LIN {X -0.173,Y -453.003,Z 1528.498,A 0.000,B 0.000,C 90.000,E1 89.714} C_DIS
LIN {X -0.072,Y -440.256,Z 1528.488,A 0.000,B 0.000,C 90.000,E1 87.879} C_DIS
LIN {X 0.196,Y -427.118,Z 1528.478,A 0.000,B 0.000,C 90.000,E1 85.988} C_DIS
LIN {X -0.048,Y -412.183,Z 1528.466,A 0.000,B 0.000,C 90.000,E1 83.856} C_DIS
LIN {X -0.163,Y -397.400,Z 1528.453,A 0.000,B 0.000,C 90.000,E1 81.659} C_DIS
LIN {X -0.079,Y -377.981,Z 1528.436,A 0.000,B 0.000,C 90.000,E1 78.522} C_DIS
LIN {X 0.029,Y -364.705,Z 1528.423,A 0.000,B 0.000,C 90.000,E1 76.172} C_DIS
LIN {X -0.004,Y -351.765,Z 1528.410,A 0.000,B 0.000,C 90.000,E1 73.795} C_DIS
LIN {X 0.181,Y -340.593,Z 1528.398,A 0.000,B 0.000,C 90.000,E1 71.638} C_DIS
LIN {X 0.080,Y -323.637,Z 1528.379,A 0.000,B 0.000,C 90.000,E1 68.230} C_DIS
LIN {X 0.151,Y -311.879,Z 1528.365,A 0.000,B 0.000,C 90.000,E1 65.665} C_DIS
LIN {X 0.063,Y -300.644,Z 1528.350,A 0.000,B 0.000,C 90.000,E1 63.076} C_DIS
LIN {X -0.152,Y -289.519,Z 1528.336,A 0.000,B 0.000,C 90.000,E1 60.461} C_DIS
LIN {X -0.057,Y -280.084,Z 1528.323,A 0.000,B 0.000,C 90.000,E1 58.074} C_DIS
LIN {X -0.116,Y -270.752,Z 1528.309,A 0.000,B 0.000,C 90.000,E1 55.674} C_DIS
LIN {X 0.046,Y -259.191,Z 1528.292,A 0.000,B 0.000,C 90.000,E1 52.477} C_DIS
LIN {X -0.016,Y -248.168,Z 1528.274,A 0.000,B 0.000,C 90.000,E1 49.256} C_DIS
LIN {X -0.099,Y -237.990,Z 1528.255,A 0.000,B 0.000,C 90.000,E1 45.972} C_DIS
LIN {X 0.109,Y -229.786,Z 1528.239,A 0.000,B 0.000,C 90.000,E1 42.933} C_DIS
LIN {X -0.028,Y -222.332,Z 1528.222,A 0.000,B 0.000,C 90.000,E1 39.930} C_DIS
LIN {X -0.117,Y -215.621,Z 1528.205,A 0.000,B 0.000,C 90.000,E1 36.870} C_DIS
LIN {X 0.019,Y -209.646,Z 1528.187,A 0.000,B 0.000,C 90.000,E1 33.706} C_DIS
LIN {X 0.009,Y -204.410,Z 1528.170,A 0.000,B 0.000,C 90.000,E1 30.541} C_DIS
LIN {X -0.017,Y -198.622,Z 1528.147,A 0.000,B 0.000,C 90.000,E1 26.539} C_DIS
LIN {X 0.049,Y -193.675,Z 1528.125,A 0.000,B 0.000,C 90.000,E1 22.461} C_DIS
LIN {X 0.035,Y -189.499,Z 1528.102,A 0.000,B 0.000,C 90.000,E1 18.362} C_DIS
LIN {X -0.030,Y -185.543,Z 1528.074,A 0.000,B 0.000,C 90.000,E1 13.411} C_DIS
LIN {X -0.030,Y -182.509,Z 1528.047,A 0.000,B 0.000,C 90.000,E1 8.398} C_DIS
LIN {X 0.030,Y -180.027,Z 1528.005,A 0.000,B 0.000,C 90.000,E1 0.802} C_DIS
LIN {X -0.035,Y -180.270,Z 1527.965,A 0.000,B 0.000,C 90.000,E1 353.628} C_DIS
LIN {X -0.026,Y -182.584,Z 1527.927,A 0.000,B 0.000,C 90.000,E1 346.881} C_DIS
LIN {X 0.077,Y -185.773,Z 1527.899,A 0.000,B 0.000,C 90.000,E1 341.819} C_DIS
LIN {X 0.047,Y -189.339,Z 1527.876,A 0.000,B 0.000,C 90.000,E1 337.667} C_DIS
LIN {X -0.030,Y -193.881,Z 1527.853,A 0.000,B 0.000,C 90.000,E1 333.563} C_DIS
LIN {X 0.100,Y -198.154,Z 1527.835,A 0.000,B 0.000,C 90.000,E1 330.255} C_DIS
LIN {X 0.094,Y -204.384,Z 1527.813,A 0.000,B 0.000,C 90.000,E1 326.215} C_DIS
LIN {X -0.012,Y -210.151,Z 1527.795,A 0.000,B 0.000,C 90.000,E1 323.050} C_DIS
LIN {X -0.059,Y -216.737,Z 1527.777,A 0.000,B 0.000,C 90.000,E1 319.908} C_DIS
LIN {X 0.005,Y -224.124,Z 1527.760,A 0.000,B 0.000,C 90.000,E1 316.782} C_DIS
LIN {X 0.043,Y -233.399,Z 1527.741,A 0.000,B 0.000,C 90.000,E1 313.338} C_DIS
LIN {X 0.126,Y -240.429,Z 1527.728,A 0.000,B 0.000,C 90.000,E1 311.067} C_DIS
LIN {X -0.137,Y -248.431,Z 1527.716,A 0.000,B 0.000,C 90.000,E1 308.910} C_DIS
LIN {X -0.087,Y -255.980,Z 1527.706,A 0.000,B 0.000,C 90.000,E1 307.076} C_DIS
LIN {X 0.099,Y -262.847,Z 1527.698,A 0.000,B 0.000,C 90.000,E1 305.598} C_DIS
LIN {X 0.009,Y -270.418,Z 1527.690,A 0.000,B 0.000,C 90.000,E1 304.199} C_DIS
LIN {X -0.047,Y -280.857,Z 1527.680,A 0.000,B 0.000,C 90.000,E1 302.467} C_DIS
LIN {X -0.034,Y -297.223,Z 1527.667,A 0.000,B 0.000,C 90.000,E1 300.079} C_DIS
LIN {X 0.000,Y -317.615,Z 1527.652,A 0.000,B 0.000,C 90.000,E1 297.436} C_DIS
LIN {X 0.091,Y -333.573,Z 1527.642,A 0.000,B 0.000,C 90.000,E1 295.540} C_DIS
LIN {X -0.050,Y -349.616,Z 1527.632,A 0.000,B 0.000,C 90.000,E1 293.770} C_DIS
LIN {X 0.136,Y -365.761,Z 1527.622,A 0.000,B 0.000,C 90.000,E1 292.025} C_DIS
LIN {X -0.085,Y -378.909,Z 1527.615,A 0.000,B 0.000,C 90.000,E1 290.663} C_DIS
LIN {X -0.010,Y -386.648,Z 1527.610,A 0.000,B 0.000,C 90.000,E1 289.812} C_DIS
LIN {X 0.039,Y -396.456,Z 1527.604,A 0.000,B 0.000,C 90.000,E1 288.671} C_DIS
LIN {X 0.076,Y -403.212,Z 1527.599,A 0.000,B 0.000,C 90.000,E1 287.819} C_DIS
LIN {X 0.046,Y -409.350,Z 1527.594,A 0.000,B 0.000,C 90.000,E1 286.985} C_DIS
LIN {X 0.081,Y -414.751,Z 1527.590,A 0.000,B 0.000,C 90.000,E1 286.150} C_DIS
LIN {X -0.242,Y -419.471,Z 1527.585,A 0.000,B 0.000,C 90.000,E1 285.371} C_DIS
LIN {X -0.119,Y -423.315,Z 1527.581,A 0.000,B 0.000,C 90.000,E1 284.537} C_DIS
LIN {X 0.035,Y -426.460,Z 1527.576,A 0.000,B 0.000,C 90.000,E1 283.703} C_DIS
LIN {X -0.057,Y -428.128,Z 1527.573,A 0.000,B 0.000,C 90.000,E1 283.175} C_DIS
LIN {X -0.138,Y -429.417,Z 1527.570,A 0.000,B 0.000,C 90.000,E1 282.647} C_DIS
LIN {X 0.213,Y -430.220,Z 1527.567,A 0.000,B 0.000,C 90.000,E1 282.063} C_DIS
LIN {X 0.150,Y -430.594,Z 1527.564,A 0.000,B 0.000,C 90.000,E1 281.535} C_DIS
LIN {X 0.091,Y -430.469,Z 1527.561,A 0.000,B 0.000,C 90.000,E1 281.007} C_DIS
LIN {X -0.045,Y -429.811,Z 1527.558,A 0.000,B 0.000,C 90.000,E1 280.489} C_DIS
LIN {X -0.103,Y -428.580,Z 1527.555,A 0.000,B 0.000,C 90.000,E1 279.962} C_DIS
LIN {X -0.167,Y -426.752,Z 1527.552,A 0.000,B 0.000,C 90.000,E1 279.434} C_DIS
LIN {X 0.112,Y -424.208,Z 1527.549,A 0.000,B 0.000,C 90.000,E1 278.859} C_DIS
LIN {X -0.042,Y -420.783,Z 1527.546,A 0.000,B 0.000,C 90.000,E1 278.341} C_DIS
LIN {X 0.111,Y -418.773,Z 1527.545,A 0.000,B 0.000,C 90.000,E1 278.049} C_DIS
LIN {X -0.068,Y -413.948,Z 1527.542,A 0.000,B 0.000,C 90.000,E1 277.530} C_DIS
LIN {X 0.070,Y -411.225,Z 1527.540,A 0.000,B 0.000,C 90.000,E1 277.239} C_DIS
LIN {X 0.063,Y -405.102,Z 1527.537,A 0.000,B 0.000,C 90.000,E1 276.720} C_DIS
LIN {X 0.110,Y -399.086,Z 1527.535,A 0.000,B 0.000,C 90.000,E1 276.258} C_DIS
LIN {X 0.027,Y -392.632,Z 1527.533,A 0.000,B 0.000,C 90.000,E1 275.853} C_DIS
LIN {X -0.142,Y -386.213,Z 1527.531,A 0.000,B 0.000,C 90.000,E1 275.511} C_DIS
LIN {X 0.106,Y -376.409,Z 1527.528,A 0.000,B 0.000,C 90.000,E1 274.992} C_DIS
LIN {X -0.035,Y -366.667,Z 1527.526,A 0.000,B 0.000,C 90.000,E1 274.588} C_DIS
LIN {X -0.112,Y -351.054,Z 1527.522,A 0.000,B 0.000,C 90.000,E1 273.955} C_DIS
LIN {X 0.037,Y -341.268,Z 1527.520,A 0.000,B 0.000,C 90.000,E1 273.555} C_DIS
LIN {X 0.087,Y -331.254,Z 1527.518,A 0.000,B 0.000,C 90.000,E1 273.212} C_DIS
LIN {X 0.142,Y -317.896,Z 1527.516,A 0.000,B 0.000,C 90.000,E1 272.808} C_DIS
LIN {X -0.021,Y -306.821,Z 1527.514,A 0.000,B 0.000,C 90.000,E1 272.579} C_DIS
LIN {X 0.106,Y -295.216,Z 1527.513,A 0.000,B 0.000,C 90.000,E1 272.350} C_DIS
LIN {X 0.098,Y -281.912,Z 1527.512,A 0.000,B 0.000,C 90.000,E1 272.178} C_DIS
LIN {X 0.024,Y -268.089,Z 1527.512,A 0.000,B 0.000,C 90.000,E1 272.121} C_DIS
LIN {X -0.008,Y -265.982,Z 1527.512,A 0.000,B 0.000,C 90.000,E1 272.121} C_DIS
LIN {X -0.027,Y -181.243,Z 1527.512,A 0.000,B 0.000,C 90.000,E1 272.121} C_DIS
LIN {X 0.068,Y -181.571,Z 1527.500,A 0.000,B 0.000,C 90.000,E1 270.057} C_DIS
LIN {X 0.056,Y -180.867,Z 1527.472,A 0.000,B 0.000,C 90.000,E1 265.008} C_DIS
LIN {X -0.067,Y -178.983,Z 1527.444,A 0.000,B 0.000,C 90.000,E1 259.982} C_DIS
LIN {X -0.056,Y -177.955,Z 1527.435,A 0.000,B 0.000,C 90.000,E1 258.285} C_DIS
LIN {X -0.037,Y -175.597,Z 1527.411,A 0.000,B 0.000,C 90.000,E1 254.031} C_DIS
LIN {X -0.023,Y -172.320,Z 1527.387,A 0.000,B 0.000,C 90.000,E1 249.752} C_DIS
LIN {X -0.045,Y -171.799,Z 1527.383,A 0.000,B 0.000,C 90.000,E1 248.901} C_DIS
LIN {X -0.007,Y -169.472,Z 1527.368,A 0.000,B 0.000,C 90.000,E1 246.305} C_DIS
LIN {X 0.048,Y -166.799,Z 1527.349,A 0.000,B 0.000,C 90.000,E1 242.820} C_DIS
LIN {X 0.043,Y -162.779,Z 1527.325,A 0.000,B 0.000,C 90.000,E1 238.456} C_DIS
LIN {X 0.019,Y -161.468,Z 1527.315,A 0.000,B 0.000,C 90.000,E1 236.707} C_DIS
LIN {X 0.059,Y -157.464,Z 1527.291,A 0.000,B 0.000,C 90.000,E1 232.271} C_DIS
LIN {X -0.008,Y -155.476,Z 1527.276,A 0.000,B 0.000,C 90.000,E1 229.622} C_DIS
LIN {X -0.074,Y -151.787,Z 1527.251,A 0.000,B 0.000,C 90.000,E1 225.162} C_DIS
LIN {X -0.061,Y -149.994,Z 1527.236,A 0.000,B 0.000,C 90.000,E1 222.447} C_DIS
LIN {X -0.030,Y -146.824,Z 1527.210,A 0.000,B 0.000,C 90.000,E1 217.890} C_DIS
LIN {X 0.076,Y -145.404,Z 1527.195,A 0.000,B 0.000,C 90.000,E1 215.105} C_DIS
LIN {X -0.007,Y -142.836,Z 1527.170,A 0.000,B 0.000,C 90.000,E1 210.541} C_DIS
LIN {X -0.077,Y -141.450,Z 1527.149,A 0.000,B 0.000,C 90.000,E1 206.873} C_DIS
LIN {X -0.036,Y -139.371,Z 1527.113,A 0.000,B 0.000,C 90.000,E1 200.355} C_DIS
LIN {X 0.038,Y -138.820,Z 1527.097,A 0.000,B 0.000,C 90.000,E1 197.528} C_DIS
LIN {X -0.005,Y -138.352,Z 1527.056,A 0.000,B 0.000,C 90.000,E1 190.074} C_DIS
LIN {X -0.033,Y -139.534,Z 1527.004,A 0.000,B 0.000,C 90.000,E1 180.745} C_DIS
LIN {X 0.060,Y -141.219,Z 1526.973,A 0.000,B 0.000,C 90.000,E1 175.122} C_DIS
LIN {X 0.019,Y -142.593,Z 1526.958,A 0.000,B 0.000,C 90.000,E1 172.356} C_DIS
LIN {X -0.027,Y -144.894,Z 1526.932,A 0.000,B 0.000,C 90.000,E1 167.757} C_DIS
LIN {X -0.074,Y -147.522,Z 1526.911,A 0.000,B 0.000,C 90.000,E1 164.102} C_DIS
LIN {X 0.000,Y -150.118,Z 1526.891,A 0.000,B 0.000,C 90.000,E1 160.423} C_DIS
LIN {X 0.012,Y -153.479,Z 1526.871,A 0.000,B 0.000,C 90.000,E1 156.794} C_DIS
LIN {X 0.076,Y -157.842,Z 1526.846,A 0.000,B 0.000,C 90.000,E1 152.281} C_DIS
LIN {X 0.032,Y -162.128,Z 1526.826,A 0.000,B 0.000,C 90.000,E1 148.742} C_DIS
LIN {X 0.011,Y -166.330,Z 1526.807,A 0.000,B 0.000,C 90.000,E1 145.229} C_DIS
LIN {X 0.018,Y -171.347,Z 1526.787,A 0.000,B 0.000,C 90.000,E1 141.743} C_DIS
LIN {X -0.054,Y -176.251,Z 1526.768,A 0.000,B 0.000,C 90.000,E1 138.324} C_DIS
LIN {X 0.064,Y -180.533,Z 1526.754,A 0.000,B 0.000,C 90.000,E1 135.729} C_DIS
LIN {X 0.043,Y -185.936,Z 1526.735,A 0.000,B 0.000,C 90.000,E1 132.366} C_DIS
LIN {X -0.021,Y -190.566,Z 1526.722,A 0.000,B 0.000,C 90.000,E1 129.886} C_DIS
LIN {X 0.009,Y -196.316,Z 1526.703,A 0.000,B 0.000,C 90.000,E1 126.583} C_DIS
LIN {X 0.087,Y -201.115,Z 1526.690,A 0.000,B 0.000,C 90.000,E1 124.119} C_DIS
LIN {X 0.060,Y -202.556,Z 1526.685,A 0.000,B 0.000,C 90.000,E1 123.293} C_DIS
LIN {X 0.042,Y -317.227,Z 1526.685,A 0.000,B 0.000,C 90.000,E1 123.293} C_DIS
LIN {X -0.114,Y -318.999,Z 1526.685,A 0.000,B 0.000,C 90.000,E1 123.293} C_DIS
LIN {X 0.003,Y -323.259,Z 1526.684,A 0.000,B 0.000,C 90.000,E1 123.086} C_DIS
LIN {X 0.122,Y -325.660,Z 1526.683,A 0.000,B 0.000,C 90.000,E1 122.880} C_DIS
LIN {X -0.092,Y -328.932,Z 1526.681,A 0.000,B 0.000,C 90.000,E1 122.546} C_DIS
LIN {X 0.077,Y -330.854,Z 1526.679,A 0.000,B 0.000,C 90.000,E1 122.212} C_DIS
LIN {X -0.033,Y -332.352,Z 1526.677,A 0.000,B 0.000,C 90.000,E1 121.926} C_DIS
LIN {X 0.120,Y -346.150,Z 1526.658,A 0.000,B 0.000,C 90.000,E1 118.487} C_DIS
LIN {X 0.015,Y -358.945,Z 1526.643,A 0.000,B 0.000,C 90.000,E1 115.771} C_DIS
LIN {X 0.137,Y -373.256,Z 1526.628,A 0.000,B 0.000,C 90.000,E1 113.078} C_DIS
LIN {X -0.112,Y -387.354,Z 1526.615,A 0.000,B 0.000,C 90.000,E1 110.791} C_DIS
LIN {X 0.084,Y -402.848,Z 1526.603,A 0.000,B 0.000,C 90.000,E1 108.489} C_DIS
LIN {X 0.165,Y -419.844,Z 1526.590,A 0.000,B 0.000,C 90.000,E1 106.260} C_DIS
LIN {X 0.012,Y -438.465,Z 1526.578,A 0.000,B 0.000,C 90.000,E1 104.120} C_DIS
LIN {X 0.039,Y -458.333,Z 1526.567,A 0.000,B 0.000,C 90.000,E1 102.063} C_DIS
LIN {X -0.147,Y -478.777,Z 1526.557,A 0.000,B 0.000,C 90.000,E1 100.197} C_DIS
LIN {X -0.161,Y -491.735,Z 1526.550,A 0.000,B 0.000,C 90.000,E1 99.095} C_DIS
LIN {X -0.031,Y -493.741,Z 1526.549,A 0.000,B 0.000,C 90.000,E1 98.859} C_DIS
LIN {X 0.099,Y -495.273,Z 1526.548,A 0.000,B 0.000,C 90.000,E1 98.624} C_DIS
LIN {X -0.061,Y -496.569,Z 1526.547,A 0.000,B 0.000,C 90.000,E1 98.398} C_DIS
LIN {X -0.149,Y -497.517,Z 1526.545,A 0.000,B 0.000,C 90.000,E1 98.163} C_DIS
LIN {X 0.114,Y -498.549,Z 1526.542,A 0.000,B 0.000,C 90.000,E1 97.644} C_DIS
LIN {X -0.110,Y -498.564,Z 1526.540,A 0.000,B 0.000,C 90.000,E1 97.182} C_DIS
LIN {X 0.166,Y -497.568,Z 1526.537,A 0.000,B 0.000,C 90.000,E1 96.663} C_DIS
LIN {X 0.084,Y -496.645,Z 1526.536,A 0.000,B 0.000,C 90.000,E1 96.429} C_DIS
LIN {X -0.052,Y -495.385,Z 1526.534,A 0.000,B 0.000,C 90.000,E1 96.201} C_DIS
LIN {X -0.132,Y -482.564,Z 1526.523,A 0.000,B 0.000,C 90.000,E1 94.245} C_DIS
LIN {X 0.031,Y -474.878,Z 1526.517,A 0.000,B 0.000,C 90.000,E1 92.980} C_DIS
LIN {X -0.148,Y -465.003,Z 1526.508,A 0.000,B 0.000,C 90.000,E1 91.489} C_DIS
LIN {X 0.185,Y -456.365,Z 1526.501,A 0.000,B 0.000,C 90.000,E1 90.172} C_DIS
LIN {X -0.066,Y -447.398,Z 1526.494,A 0.000,B 0.000,C 90.000,E1 88.912} C_DIS
LIN {X 0.019,Y -438.249,Z 1526.487,A 0.000,B 0.000,C 90.000,E1 87.593} C_DIS
LIN {X -0.160,Y -425.115,Z 1526.476,A 0.000,B 0.000,C 90.000,E1 85.755} C_DIS
LIN {X -0.064,Y -410.273,Z 1526.464,A 0.000,B 0.000,C 90.000,E1 83.571} C_DIS
LIN {X -0.154,Y -393.712,Z 1526.450,A 0.000,B 0.000,C 90.000,E1 81.084} C_DIS
LIN {X -0.141,Y -376.233,Z 1526.434,A 0.000,B 0.000,C 90.000,E1 78.229} C_DIS
LIN {X -0.074,Y -363.041,Z 1526.422,A 0.000,B 0.000,C 90.000,E1 75.880} C_DIS
LIN {X -0.086,Y -351.730,Z 1526.410,A 0.000,B 0.000,C 90.000,E1 73.795} C_DIS
LIN {X 0.101,Y -340.554,Z 1526.398,A 0.000,B 0.000,C 90.000,E1 71.638} C_DIS
LIN {X 0.002,Y -323.597,Z 1526.379,A 0.000,B 0.000,C 90.000,E1 68.230} C_DIS
LIN {X -0.002,Y -310.395,Z 1526.363,A 0.000,B 0.000,C 90.000,E1 65.357} C_DIS
LIN {X 0.011,Y -299.185,Z 1526.349,A 0.000,B 0.000,C 90.000,E1 62.743} C_DIS
LIN {X 0.018,Y -288.141,Z 1526.334,A 0.000,B 0.000,C 90.000,E1 60.078} C_DIS
LIN {X -0.019,Y -278.750,Z 1526.321,A 0.000,B 0.000,C 90.000,E1 57.709} C_DIS
LIN {X -0.170,Y -268.179,Z 1526.305,A 0.000,B 0.000,C 90.000,E1 54.975} C_DIS
LIN {X 0.030,Y -258.026,Z 1526.290,A 0.000,B 0.000,C 90.000,E1 52.110} C_DIS
LIN {X 0.102,Y -247.111,Z 1526.271,A 0.000,B 0.000,C 90.000,E1 48.852} C_DIS
LIN {X -0.152,Y -238.144,Z 1526.255,A 0.000,B 0.000,C 90.000,E1 45.972} C_DIS
LIN {X 0.068,Y -229.958,Z 1526.239,A 0.000,B 0.000,C 90.000,E1 42.933} C_DIS
LIN {X -0.064,Y -222.521,Z 1526.222,A 0.000,B 0.000,C 90.000,E1 39.930} C_DIS
LIN {X 0.026,Y -215.851,Z 1526.205,A 0.000,B 0.000,C 90.000,E1 36.824} C_DIS
LIN {X -0.004,Y -209.917,Z 1526.187,A 0.000,B 0.000,C 90.000,E1 33.706} C_DIS
LIN {X -0.006,Y -204.679,Z 1526.170,A 0.000,B 0.000,C 90.000,E1 30.541} C_DIS
LIN {X -0.024,Y -198.893,Z 1526.147,A 0.000,B 0.000,C 90.000,E1 26.539} C_DIS
LIN {X 0.051,Y -193.952,Z 1526.125,A 0.000,B 0.000,C 90.000,E1 22.461} C_DIS
LIN {X 0.045,Y -189.771,Z 1526.102,A 0.000,B 0.000,C 90.000,E1 18.362} C_DIS
LIN {X -0.010,Y -185.781,Z 1526.074,A 0.000,B 0.000,C 90.000,E1 13.411} C_DIS
LIN {X -0.092,Y -182.340,Z 1526.042,A 0.000,B 0.000,C 90.000,E1 7.587} C_DIS
LIN {X -0.032,Y -180.199,Z 1525.997,A 0.000,B 0.000,C 90.000,E1 359.542} C_DIS
LIN {X 0.050,Y -180.694,Z 1525.960,A 0.000,B 0.000,C 90.000,E1 352.761} C_DIS
LIN {X -0.023,Y -183.276,Z 1525.922,A 0.000,B 0.000,C 90.000,E1 346.047} C_DIS
LIN {X -0.068,Y -186.654,Z 1525.895,A 0.000,B 0.000,C 90.000,E1 341.040} C_DIS
LIN {X -0.012,Y -190.368,Z 1525.871,A 0.000,B 0.000,C 90.000,E1 336.869} C_DIS
LIN {X 0.020,Y -195.079,Z 1525.849,A 0.000,B 0.000,C 90.000,E1 332.743} C_DIS
LIN {X 0.050,Y -200.690,Z 1525.826,A 0.000,B 0.000,C 90.000,E1 328.663} C_DIS
LIN {X -0.041,Y -205.912,Z 1525.808,A 0.000,B 0.000,C 90.000,E1 325.468} C_DIS
LIN {X 0.008,Y -211.870,Z 1525.790,A 0.000,B 0.000,C 90.000,E1 322.271} C_DIS
LIN {X -0.026,Y -218.636,Z 1525.773,A 0.000,B 0.000,C 90.000,E1 319.138} C_DIS
LIN {X 0.011,Y -227.200,Z 1525.754,A 0.000,B 0.000,C 90.000,E1 315.648} C_DIS
LIN {X 0.029,Y -235.753,Z 1525.737,A 0.000,B 0.000,C 90.000,E1 312.609} C_DIS
LIN {X -0.008,Y -243.086,Z 1525.724,A 0.000,B 0.000,C 90.000,E1 310.378} C_DIS
LIN {X -0.032,Y -251.392,Z 1525.712,A 0.000,B 0.000,C 90.000,E1 308.177} C_DIS
LIN {X 0.041,Y -257.616,Z 1525.704,A 0.000,B 0.000,C 90.000,E1 306.710} C_DIS
LIN {X -0.070,Y -266.486,Z 1525.694,A 0.000,B 0.000,C 90.000,E1 304.945} C_DIS
LIN {X 0.035,Y -276.442,Z 1525.684,A 0.000,B 0.000,C 90.000,E1 303.166} C_DIS
LIN {X -0.085,Y -287.502,Z 1525.675,A 0.000,B 0.000,C 90.000,E1 301.465} C_DIS
LIN {X -0.008,Y -309.538,Z 1525.658,A 0.000,B 0.000,C 90.000,E1 298.437} C_DIS
LIN {X -0.082,Y -330.555,Z 1525.644,A 0.000,B 0.000,C 90.000,E1 295.924} C_DIS
LIN {X 0.157,Y -349.448,Z 1525.632,A 0.000,B 0.000,C 90.000,E1 293.770} C_DIS
LIN {X 0.030,Y -365.620,Z 1525.623,A 0.000,B 0.000,C 90.000,E1 292.078} C_DIS
LIN {X 0.051,Y -378.769,Z 1525.615,A 0.000,B 0.000,C 90.000,E1 290.684} C_DIS
LIN {X -0.088,Y -386.496,Z 1525.610,A 0.000,B 0.000,C 90.000,E1 289.866} C_DIS
LIN {X -0.088,Y -393.952,Z 1525.606,A 0.000,B 0.000,C 90.000,E1 289.014} C_DIS
LIN {X -0.212,Y -401.000,Z 1525.601,A 0.000,B 0.000,C 90.000,E1 288.181} C_DIS
LIN {X -0.141,Y -407.348,Z 1525.596,A 0.000,B 0.000,C 90.000,E1 287.330} C_DIS
LIN {X -0.138,Y -413.082,Z 1525.592,A 0.000,B 0.000,C 90.000,E1 286.496} C_DIS
LIN {X 0.203,Y -416.536,Z 1525.589,A 0.000,B 0.000,C 90.000,E1 285.898} C_DIS
LIN {X 0.053,Y -419.609,Z 1525.585,A 0.000,B 0.000,C 90.000,E1 285.371} C_DIS
LIN {X 0.180,Y -423.507,Z 1525.581,A 0.000,B 0.000,C 90.000,E1 284.537} C_DIS
LIN {X 0.077,Y -425.750,Z 1525.578,A 0.000,B 0.000,C 90.000,E1 284.008} C_DIS
LIN {X -0.163,Y -428.421,Z 1525.573,A 0.000,B 0.000,C 90.000,E1 283.231} C_DIS
LIN {X 0.176,Y -429.747,Z 1525.570,A 0.000,B 0.000,C 90.000,E1 282.647} C_DIS
LIN {X 0.108,Y -430.664,Z 1525.567,A 0.000,B 0.000,C 90.000,E1 282.119} C_DIS
LIN {X 0.047,Y -431.055,Z 1525.564,A 0.000,B 0.000,C 90.000,E1 281.591} C_DIS
LIN {X -0.093,Y -431.020,Z 1525.561,A 0.000,B 0.000,C 90.000,E1 281.074} C_DIS
LIN {X -0.146,Y -430.406,Z 1525.558,A 0.000,B 0.000,C 90.000,E1 280.546} C_DIS
LIN {X 0.222,Y -429.247,Z 1525.556,A 0.000,B 0.000,C 90.000,E1 279.962} C_DIS
LIN {X 0.091,Y -427.504,Z 1525.552,A 0.000,B 0.000,C 90.000,E1 279.443} C_DIS
LIN {X 0.022,Y -425.035,Z 1525.550,A 0.000,B 0.000,C 90.000,E1 278.916} C_DIS
LIN {X -0.127,Y -421.724,Z 1525.547,A 0.000,B 0.000,C 90.000,E1 278.398} C_DIS
LIN {X 0.028,Y -419.779,Z 1525.545,A 0.000,B 0.000,C 90.000,E1 278.106} C_DIS
LIN {X -0.144,Y -415.081,Z 1525.542,A 0.000,B 0.000,C 90.000,E1 277.587} C_DIS
LIN {X -0.223,Y -409.526,Z 1525.539,A 0.000,B 0.000,C 90.000,E1 277.068} C_DIS
LIN {X 0.002,Y -403.518,Z 1525.536,A 0.000,B 0.000,C 90.000,E1 276.549} C_DIS
LIN {X 0.155,Y -397.292,Z 1525.534,A 0.000,B 0.000,C 90.000,E1 276.087} C_DIS
LIN {X -0.180,Y -390.890,Z 1525.532,A 0.000,B 0.000,C 90.000,E1 275.739} C_DIS
LIN {X 0.156,Y -384.382,Z 1525.530,A 0.000,B 0.000,C 90.000,E1 275.334} C_DIS
LIN {X 0.051,Y -374.399,Z 1525.527,A 0.000,B 0.000,C 90.000,E1 274.878} C_DIS
LIN {X -0.149,Y -358.593,Z 1525.523,A 0.000,B 0.000,C 90.000,E1 274.245} C_DIS
LIN {X -0.071,Y -345.966,Z 1525.521,A 0.000,B 0.000,C 90.000,E1 273.726} C_DIS
LIN {X -0.158,Y -335.860,Z 1525.519,A 0.000,B 0.000,C 90.000,E1 273.383} C_DIS
LIN {X 0.153,Y -322.648,Z 1525.516,A 0.000,B 0.000,C 90.000,E1 272.922} C_DIS
LIN {X -0.096,Y -311.980,Z 1525.515,A 0.000,B 0.000,C 90.000,E1 272.694} C_DIS
LIN {X -0.107,Y -300.382,Z 1525.514,A 0.000,B 0.000,C 90.000,E1 272.465} C_DIS
LIN {X 0.139,Y -287.899,Z 1525.513,A 0.000,B 0.000,C 90.000,E1 272.236} C_DIS
LIN {X -0.076,Y -276.839,Z 1525.512,A 0.000,B 0.000,C 90.000,E1 272.178} C_DIS
LIN {X 0.005,Y -265.525,Z 1525.512,A 0.000,B 0.000,C 90.000,E1 272.121} C_DIS
LIN {X -0.018,Y -181.244,Z 1525.512,A 0.000,B 0.000,C 90.000,E1 272.121} C_DIS
LIN {X -0.082,Y -181.572,Z 1525.500,A 0.000,B 0.000,C 90.000,E1 270.115} C_DIS
LIN {X 0.086,Y -180.870,Z 1525.472,A 0.000,B 0.000,C 90.000,E1 265.008} C_DIS
LIN {X -0.037,Y -178.985,Z 1525.444,A 0.000,B 0.000,C 90.000,E1 259.982} C_DIS
LIN {X -0.025,Y -177.962,Z 1525.435,A 0.000,B 0.000,C 90.000,E1 258.285} C_DIS
LIN {X -0.006,Y -175.604,Z 1525.411,A 0.000,B 0.000,C 90.000,E1 254.031} C_DIS
LIN {X 0.006,Y -172.328,Z 1525.388,A 0.000,B 0.000,C 90.000,E1 249.752} C_DIS
LIN {X -0.015,Y -171.804,Z 1525.383,A 0.000,B 0.000,C 90.000,E1 248.901} C_DIS
LIN {X -0.008,Y -170.264,Z 1525.373,A 0.000,B 0.000,C 90.000,E1 247.177} C_DIS
LIN {X -0.071,Y -166.807,Z 1525.349,A 0.000,B 0.000,C 90.000,E1 242.871} C_DIS
LIN {X 0.072,Y -162.788,Z 1525.325,A 0.000,B 0.000,C 90.000,E1 238.456} C_DIS
LIN {X 0.047,Y -161.476,Z 1525.315,A 0.000,B 0.000,C 90.000,E1 236.707} C_DIS
LIN {X -0.037,Y -157.471,Z 1525.291,A 0.000,B 0.000,C 90.000,E1 232.316} C_DIS
LIN {X 0.020,Y -155.486,Z 1525.276,A 0.000,B 0.000,C 90.000,E1 229.622} C_DIS
LIN {X -0.048,Y -151.794,Z 1525.251,A 0.000,B 0.000,C 90.000,E1 225.162} C_DIS
LIN {X -0.034,Y -150.003,Z 1525.236,A 0.000,B 0.000,C 90.000,E1 222.447} C_DIS
LIN {X -0.003,Y -146.830,Z 1525.210,A 0.000,B 0.000,C 90.000,E1 217.890} C_DIS
LIN {X -0.016,Y -145.411,Z 1525.195,A 0.000,B 0.000,C 90.000,E1 215.152} C_DIS
LIN {X 0.019,Y -142.841,Z 1525.170,A 0.000,B 0.000,C 90.000,E1 210.541} C_DIS
LIN {X -0.050,Y -141.455,Z 1525.149,A 0.000,B 0.000,C 90.000,E1 206.873} C_DIS
LIN {X -0.011,Y -139.373,Z 1525.113,A 0.000,B 0.000,C 90.000,E1 200.355} C_DIS
LIN {X -0.068,Y -138.822,Z 1525.098,A 0.000,B 0.000,C 90.000,E1 197.583} C_DIS
LIN {X 0.020,Y -138.353,Z 1525.056,A 0.000,B 0.000,C 90.000,E1 190.074} C_DIS
LIN {X -0.007,Y -139.533,Z 1525.004,A 0.000,B 0.000,C 90.000,E1 180.745} C_DIS
LIN {X -0.054,Y -141.214,Z 1524.973,A 0.000,B 0.000,C 90.000,E1 175.179} C_DIS
LIN {X 0.046,Y -142.588,Z 1524.958,A 0.000,B 0.000,C 90.000,E1 172.356} C_DIS
LIN {X 0.000,Y -144.887,Z 1524.932,A 0.000,B 0.000,C 90.000,E1 167.757} C_DIS
LIN {X -0.047,Y -147.515,Z 1524.912,A 0.000,B 0.000,C 90.000,E1 164.102} C_DIS
LIN {X 0.027,Y -150.109,Z 1524.891,A 0.000,B 0.000,C 90.000,E1 160.423} C_DIS
LIN {X 0.040,Y -153.468,Z 1524.871,A 0.000,B 0.000,C 90.000,E1 156.794} C_DIS
LIN {X 0.031,Y -157.832,Z 1524.846,A 0.000,B 0.000,C 90.000,E1 152.308} C_DIS
LIN {X 0.060,Y -162.115,Z 1524.826,A 0.000,B 0.000,C 90.000,E1 148.742} C_DIS
LIN {X -0.054,Y -166.317,Z 1524.807,A 0.000,B 0.000,C 90.000,E1 145.261} C_DIS
LIN {X 0.048,Y -171.335,Z 1524.788,A 0.000,B 0.000,C 90.000,E1 141.743} C_DIS
LIN {X -0.024,Y -176.236,Z 1524.768,A 0.000,B 0.000,C 90.000,E1 138.324} C_DIS
LIN {X 0.095,Y -180.516,Z 1524.754,A 0.000,B 0.000,C 90.000,E1 135.729} C_DIS
LIN {X 0.075,Y -185.919,Z 1524.735,A 0.000,B 0.000,C 90.000,E1 132.366} C_DIS
LIN {X 0.011,Y -190.548,Z 1524.722,A 0.000,B 0.000,C 90.000,E1 129.886} C_DIS
LIN {X 0.042,Y -196.299,Z 1524.703,A 0.000,B 0.000,C 90.000,E1 126.583} C_DIS
LIN {X 0.120,Y -201.098,Z 1524.690,A 0.000,B 0.000,C 90.000,E1 124.119} C_DIS
LIN {X -0.119,Y -202.506,Z 1524.685,A 0.000,B 0.000,C 90.000,E1 123.372} C_DIS
LIN {X 0.217,Y -317.322,Z 1524.685,A 0.000,B 0.000,C 90.000,E1 123.293} C_DIS
LIN {X -0.062,Y -319.730,Z 1524.685,A 0.000,B 0.000,C 90.000,E1 123.293} C_DIS
LIN {X 0.055,Y -323.481,Z 1524.684,A 0.000,B 0.000,C 90.000,E1 123.086} C_DIS
LIN {X 0.175,Y -325.777,Z 1524.683,A 0.000,B 0.000,C 90.000,E1 122.880} C_DIS
LIN {X -0.039,Y -328.959,Z 1524.681,A 0.000,B 0.000,C 90.000,E1 122.546} C_DIS
LIN {X 0.097,Y -330.873,Z 1524.679,A 0.000,B 0.000,C 90.000,E1 122.212} C_DIS
LIN {X -0.049,Y -332.363,Z 1524.677,A 0.000,B 0.000,C 90.000,E1 121.926} C_DIS
LIN {X -0.059,Y -344.809,Z 1524.660,A 0.000,B 0.000,C 90.000,E1 118.821} C_DIS
LIN {X 0.123,Y -357.440,Z 1524.645,A 0.000,B 0.000,C 90.000,E1 116.052} C_DIS
LIN {X 0.024,Y -371.581,Z 1524.630,A 0.000,B 0.000,C 90.000,E1 113.387} C_DIS
LIN {X 0.088,Y -385.514,Z 1524.617,A 0.000,B 0.000,C 90.000,E1 111.046} C_DIS
LIN {X 0.001,Y -400.829,Z 1524.604,A 0.000,B 0.000,C 90.000,E1 108.779} C_DIS
LIN {X 0.019,Y -417.634,Z 1524.592,A 0.000,B 0.000,C 90.000,E1 106.551} C_DIS
LIN {X 0.222,Y -436.047,Z 1524.580,A 0.000,B 0.000,C 90.000,E1 104.356} C_DIS
LIN {X 0.096,Y -455.830,Z 1524.568,A 0.000,B 0.000,C 90.000,E1 102.299} C_DIS
LIN {X -0.162,Y -476.207,Z 1524.558,A 0.000,B 0.000,C 90.000,E1 100.423} C_DIS
LIN {X -0.182,Y -491.721,Z 1524.550,A 0.000,B 0.000,C 90.000,E1 99.095} C_DIS
LIN {X -0.059,Y -493.713,Z 1524.549,A 0.000,B 0.000,C 90.000,E1 98.859} C_DIS
LIN {X 0.064,Y -495.234,Z 1524.548,A 0.000,B 0.000,C 90.000,E1 98.624} C_DIS
LIN {X -0.097,Y -496.515,Z 1524.547,A 0.000,B 0.000,C 90.000,E1 98.398} C_DIS
LIN {X -0.184,Y -497.451,Z 1524.545,A 0.000,B 0.000,C 90.000,E1 98.163} C_DIS
LIN {X 0.079,Y -498.463,Z 1524.542,A 0.000,B 0.000,C 90.000,E1 97.644} C_DIS
LIN {X -0.146,Y -498.459,Z 1524.540,A 0.000,B 0.000,C 90.000,E1 97.182} C_DIS
LIN {X 0.129,Y -497.444,Z 1524.537,A 0.000,B 0.000,C 90.000,E1 96.663} C_DIS
LIN {X 0.047,Y -496.510,Z 1524.536,A 0.000,B 0.000,C 90.000,E1 96.429} C_DIS
LIN {X -0.089,Y -495.235,Z 1524.534,A 0.000,B 0.000,C 90.000,E1 96.201} C_DIS
LIN {X -0.006,Y -483.924,Z 1524.525,A 0.000,B 0.000,C 90.000,E1 94.473} C_DIS
LIN {X -0.004,Y -474.725,Z 1524.517,A 0.000,B 0.000,C 90.000,E1 92.980} C_DIS
LIN {X 0.016,Y -466.534,Z 1524.510,A 0.000,B 0.000,C 90.000,E1 91.718} C_DIS
LIN {X -0.094,Y -457.981,Z 1524.502,A 0.000,B 0.000,C 90.000,E1 90.458} C_DIS
LIN {X 0.137,Y -449.089,Z 1524.495,A 0.000,B 0.000,C 90.000,E1 89.141} C_DIS
LIN {X -0.203,Y -440.013,Z 1524.488,A 0.000,B 0.000,C 90.000,E1 87.879} C_DIS
LIN {X -0.075,Y -428.787,Z 1524.479,A 0.000,B 0.000,C 90.000,E1 86.274} C_DIS
LIN {X 0.015,Y -415.746,Z 1524.469,A 0.000,B 0.000,C 90.000,E1 84.375} C_DIS
LIN {X 0.074,Y -406.525,Z 1524.461,A 0.000,B 0.000,C 90.000,E1 82.996} C_DIS
LIN {X -0.058,Y -390.096,Z 1524.447,A 0.000,B 0.000,C 90.000,E1 80.500} C_DIS
LIN {X -0.145,Y -369.575,Z 1524.428,A 0.000,B 0.000,C 90.000,E1 77.061} C_DIS
LIN {X -0.060,Y -356.569,Z 1524.415,A 0.000,B 0.000,C 90.000,E1 74.685} C_DIS
LIN {X 0.127,Y -345.338,Z 1524.403,A 0.000,B 0.000,C 90.000,E1 72.543} C_DIS
LIN {X -0.071,Y -331.094,Z 1524.388,A 0.000,B 0.000,C 90.000,E1 69.806} C_DIS
LIN {X -0.047,Y -319.131,Z 1524.374,A 0.000,B 0.000,C 90.000,E1 67.283} C_DIS
LIN {X -0.168,Y -306.106,Z 1524.358,A 0.000,B 0.000,C 90.000,E1 64.409} C_DIS
LIN {X -0.127,Y -296.382,Z 1524.345,A 0.000,B 0.000,C 90.000,E1 62.103} C_DIS
LIN {X -0.045,Y -285.460,Z 1524.330,A 0.000,B 0.000,C 90.000,E1 59.410} C_DIS
LIN {X -0.136,Y -276.149,Z 1524.317,A 0.000,B 0.000,C 90.000,E1 57.041} C_DIS
LIN {X -0.127,Y -264.459,Z 1524.299,A 0.000,B 0.000,C 90.000,E1 53.909} C_DIS
LIN {X 0.007,Y -253.232,Z 1524.282,A 0.000,B 0.000,C 90.000,E1 50.678} C_DIS
LIN {X 0.075,Y -242.686,Z 1524.263,A 0.000,B 0.000,C 90.000,E1 47.391} C_DIS
LIN {X 0.057,Y -234.133,Z 1524.247,A 0.000,B 0.000,C 90.000,E1 44.433} C_DIS
LIN {X 0.010,Y -226.369,Z 1524.230,A 0.000,B 0.000,C 90.000,E1 41.434} C_DIS
LIN {X -0.018,Y -219.339,Z 1524.213,A 0.000,B 0.000,C 90.000,E1 38.382} C_DIS
LIN {X 0.038,Y -213.066,Z 1524.196,A 0.000,B 0.000,C 90.000,E1 35.264} C_DIS
LIN {X -0.010,Y -207.497,Z 1524.178,A 0.000,B 0.000,C 90.000,E1 32.133} C_DIS
LIN {X -0.021,Y -201.414,Z 1524.156,A 0.000,B 0.000,C 90.000,E1 28.153} C_DIS
LIN {X -0.063,Y -196.107,Z 1524.134,A 0.000,B 0.000,C 90.000,E1 24.131} C_DIS
LIN {X -0.050,Y -191.619,Z 1524.111,A 0.000,B 0.000,C 90.000,E1 20.047} C_DIS
LIN {X 0.061,Y -187.282,Z 1524.084,A 0.000,B 0.000,C 90.000,E1 15.064} C_DIS
LIN {X 0.044,Y -183.892,Z 1524.056,A 0.000,B 0.000,C 90.000,E1 10.074} C_DIS
LIN {X -0.026,Y -181.074,Z 1524.019,A 0.000,B 0.000,C 90.000,E1 3.383} C_DIS
LIN {X 0.043,Y -180.544,Z 1523.974,A 0.000,B 0.000,C 90.000,E1 355.298} C_DIS
LIN {X 0.086,Y -182.656,Z 1523.932,A 0.000,B 0.000,C 90.000,E1 347.701} C_DIS
LIN {X -0.085,Y -185.635,Z 1523.904,A 0.000,B 0.000,C 90.000,E1 342.725} C_DIS
LIN {X -0.013,Y -188.992,Z 1523.881,A 0.000,B 0.000,C 90.000,E1 338.539} C_DIS
LIN {X -0.013,Y -193.287,Z 1523.858,A 0.000,B 0.000,C 90.000,E1 334.409} C_DIS
LIN {X -0.061,Y -198.503,Z 1523.835,A 0.000,B 0.000,C 90.000,E1 330.333} C_DIS
LIN {X -0.035,Y -203.371,Z 1523.817,A 0.000,B 0.000,C 90.000,E1 327.089} C_DIS
LIN {X 0.054,Y -208.932,Z 1523.799,A 0.000,B 0.000,C 90.000,E1 323.863} C_DIS
LIN {X -0.027,Y -215.276,Z 1523.782,A 0.000,B 0.000,C 90.000,E1 320.723} C_DIS
LIN {X 0.005,Y -222.435,Z 1523.764,A 0.000,B 0.000,C 90.000,E1 317.595} C_DIS
LIN {X -0.010,Y -231.449,Z 1523.745,A 0.000,B 0.000,C 90.000,E1 314.150} C_DIS
LIN {X -0.008,Y -239.419,Z 1523.731,A 0.000,B 0.000,C 90.000,E1 311.515} C_DIS
LIN {X 0.052,Y -247.218,Z 1523.718,A 0.000,B 0.000,C 90.000,E1 309.277} C_DIS
LIN {X 0.094,Y -254.475,Z 1523.708,A 0.000,B 0.000,C 90.000,E1 307.443} C_DIS
LIN {X 0.053,Y -261.038,Z 1523.700,A 0.000,B 0.000,C 90.000,E1 306.011} C_DIS
LIN {X -0.061,Y -268.334,Z 1523.692,A 0.000,B 0.000,C 90.000,E1 304.612} C_DIS
LIN {X 0.074,Y -278.456,Z 1523.682,A 0.000,B 0.000,C 90.000,E1 302.832} C_DIS
LIN {X 0.001,Y -289.658,Z 1523.673,A 0.000,B 0.000,C 90.000,E1 301.131} C_DIS
LIN {X -0.155,Y -309.328,Z 1523.658,A 0.000,B 0.000,C 90.000,E1 298.487} C_DIS
LIN {X -0.024,Y -330.476,Z 1523.644,A 0.000,B 0.000,C 90.000,E1 295.924} C_DIS
LIN {X 0.056,Y -349.249,Z 1523.632,A 0.000,B 0.000,C 90.000,E1 293.823} C_DIS
LIN {X -0.117,Y -365.339,Z 1523.623,A 0.000,B 0.000,C 90.000,E1 292.153} C_DIS
LIN {X 0.044,Y -378.519,Z 1523.615,A 0.000,B 0.000,C 90.000,E1 290.737} C_DIS
LIN {X 0.131,Y -386.235,Z 1523.611,A 0.000,B 0.000,C 90.000,E1 289.885} C_DIS
LIN {X 0.120,Y -393.767,Z 1523.606,A 0.000,B 0.000,C 90.000,E1 289.033} C_DIS
LIN {X 0.127,Y -400.849,Z 1523.601,A 0.000,B 0.000,C 90.000,E1 288.181} C_DIS
LIN {X 0.082,Y -407.273,Z 1523.596,A 0.000,B 0.000,C 90.000,E1 287.347} C_DIS
LIN {X 0.210,Y -413.080,Z 1523.592,A 0.000,B 0.000,C 90.000,E1 286.496} C_DIS
LIN {X -0.125,Y -418.169,Z 1523.587,A 0.000,B 0.000,C 90.000,E1 285.717} C_DIS
LIN {X -0.129,Y -422.431,Z 1523.583,A 0.000,B 0.000,C 90.000,E1 284.898} C_DIS
LIN {X 0.024,Y -425.952,Z 1523.578,A 0.000,B 0.000,C 90.000,E1 284.064} C_DIS
LIN {X 0.103,Y -428.695,Z 1523.574,A 0.000,B 0.000,C 90.000,E1 283.244} C_DIS
LIN {X 0.029,Y -430.065,Z 1523.571,A 0.000,B 0.000,C 90.000,E1 282.715} C_DIS
LIN {X -0.035,Y -431.037,Z 1523.568,A 0.000,B 0.000,C 90.000,E1 282.187} C_DIS
LIN {X -0.091,Y -431.555,Z 1523.565,A 0.000,B 0.000,C 90.000,E1 281.658} C_DIS
LIN {X -0.143,Y -431.579,Z 1523.562,A 0.000,B 0.000,C 90.000,E1 281.130} C_DIS
LIN {X -0.193,Y -431.048,Z 1523.559,A 0.000,B 0.000,C 90.000,E1 280.602} C_DIS
LIN {X 0.178,Y -429.995,Z 1523.556,A 0.000,B 0.000,C 90.000,E1 280.018} C_DIS
LIN {X 0.049,Y -428.268,Z 1523.553,A 0.000,B 0.000,C 90.000,E1 279.500} C_DIS
LIN {X -0.015,Y -425.864,Z 1523.550,A 0.000,B 0.000,C 90.000,E1 278.973} C_DIS
LIN {X 0.088,Y -424.429,Z 1523.548,A 0.000,B 0.000,C 90.000,E1 278.690} C_DIS
LIN {X -0.003,Y -420.821,Z 1523.545,A 0.000,B 0.000,C 90.000,E1 278.163} C_DIS
LIN {X -0.170,Y -416.222,Z 1523.542,A 0.000,B 0.000,C 90.000,E1 277.644} C_DIS
LIN {X 0.122,Y -410.739,Z 1523.539,A 0.000,B 0.000,C 90.000,E1 277.068} C_DIS
LIN {X -0.129,Y -404.726,Z 1523.537,A 0.000,B 0.000,C 90.000,E1 276.606} C_DIS
LIN {X -0.002,Y -398.530,Z 1523.534,A 0.000,B 0.000,C 90.000,E1 276.144} C_DIS
LIN {X 0.029,Y -392.136,Z 1523.532,A 0.000,B 0.000,C 90.000,E1 275.739} C_DIS
LIN {X -0.041,Y -385.646,Z 1523.530,A 0.000,B 0.000,C 90.000,E1 275.391} C_DIS
LIN {X -0.117,Y -375.802,Z 1523.527,A 0.000,B 0.000,C 90.000,E1 274.935} C_DIS
LIN {X 0.039,Y -359.942,Z 1523.524,A 0.000,B 0.000,C 90.000,E1 274.245} C_DIS
LIN {X 0.097,Y -347.275,Z 1523.521,A 0.000,B 0.000,C 90.000,E1 273.726} C_DIS
LIN {X -0.008,Y -337.107,Z 1523.519,A 0.000,B 0.000,C 90.000,E1 273.383} C_DIS
LIN {X -0.021,Y -324.031,Z 1523.516,A 0.000,B 0.000,C 90.000,E1 272.980} C_DIS
LIN {X 0.068,Y -313.867,Z 1523.515,A 0.000,B 0.000,C 90.000,E1 272.694} C_DIS
LIN {X 0.030,Y -302.489,Z 1523.514,A 0.000,B 0.000,C 90.000,E1 272.465} C_DIS
LIN {X -0.033,Y -290.317,Z 1523.513,A 0.000,B 0.000,C 90.000,E1 272.293} C_DIS
LIN {X 0.015,Y -280.253,Z 1523.512,A 0.000,B 0.000,C 90.000,E1 272.178} C_DIS
LIN {X 0.052,Y -269.401,Z 1523.512,A 0.000,B 0.000,C 90.000,E1 272.121} C_DIS
LIN {X 0.009,Y -262.863,Z 1523.512,A 0.000,B 0.000,C 90.000,E1 272.121} C_DIS
LIN {X -0.022,Y -181.243,Z 1523.512,A 0.000,B 0.000,C 90.000,E1 272.121} C_DIS
LIN {X -0.080,Y -181.578,Z 1523.502,A 0.000,B 0.000,C 90.000,E1 270.401} C_DIS
LIN {X 0.077,Y -180.904,Z 1523.474,A 0.000,B 0.000,C 90.000,E1 265.298} C_DIS
LIN {X 0.027,Y -180.255,Z 1523.465,A 0.000,B 0.000,C 90.000,E1 263.628} C_DIS
LIN {X 0.046,Y -178.746,Z 1523.441,A 0.000,B 0.000,C 90.000,E1 259.398} C_DIS
LIN {X -0.056,Y -175.793,Z 1523.413,A 0.000,B 0.000,C 90.000,E1 254.338} C_DIS
LIN {X -0.062,Y -171.978,Z 1523.384,A 0.000,B 0.000,C 90.000,E1 249.209} C_DIS
LIN {X -0.024,Y -171.381,Z 1523.380,A 0.000,B 0.000,C 90.000,E1 248.337} C_DIS
LIN {X -0.038,Y -167.626,Z 1523.356,A 0.000,B 0.000,C 90.000,E1 244.024} C_DIS
LIN {X -0.023,Y -166.280,Z 1523.346,A 0.000,B 0.000,C 90.000,E1 242.281} C_DIS
LIN {X -0.028,Y -163.030,Z 1523.327,A 0.000,B 0.000,C 90.000,E1 238.791} C_DIS
LIN {X 0.024,Y -160.958,Z 1523.312,A 0.000,B 0.000,C 90.000,E1 236.135} C_DIS
LIN {X 0.007,Y -157.712,Z 1523.292,A 0.000,B 0.000,C 90.000,E1 232.603} C_DIS
LIN {X 0.071,Y -155.752,Z 1523.277,A 0.000,B 0.000,C 90.000,E1 229.908} C_DIS
LIN {X 0.016,Y -152.009,Z 1523.253,A 0.000,B 0.000,C 90.000,E1 225.445} C_DIS
LIN {X -0.074,Y -150.254,Z 1523.237,A 0.000,B 0.000,C 90.000,E1 222.771} C_DIS
LIN {X 0.061,Y -147.011,Z 1523.212,A 0.000,B 0.000,C 90.000,E1 218.177} C_DIS
LIN {X 0.050,Y -145.594,Z 1523.197,A 0.000,B 0.000,C 90.000,E1 215.438} C_DIS
LIN {X -0.030,Y -142.981,Z 1523.172,A 0.000,B 0.000,C 90.000,E1 210.875} C_DIS
LIN {X -0.030,Y -141.608,Z 1523.151,A 0.000,B 0.000,C 90.000,E1 207.180} C_DIS
LIN {X 0.012,Y -139.426,Z 1523.115,A 0.000,B 0.000,C 90.000,E1 200.663} C_DIS
LIN {X 0.063,Y -139.155,Z 1523.104,A 0.000,B 0.000,C 90.000,E1 198.779} C_DIS
LIN {X -0.051,Y -138.343,Z 1523.058,A 0.000,B 0.000,C 90.000,E1 190.423} C_DIS
LIN {X -0.069,Y -139.483,Z 1523.006,A 0.000,B 0.000,C 90.000,E1 181.088} C_DIS
LIN {X 0.012,Y -141.077,Z 1522.975,A 0.000,B 0.000,C 90.000,E1 175.469} C_DIS
LIN {X -0.035,Y -142.453,Z 1522.959,A 0.000,B 0.000,C 90.000,E1 172.704} C_DIS
LIN {X 0.055,Y -144.695,Z 1522.934,A 0.000,B 0.000,C 90.000,E1 168.049} C_DIS
LIN {X 0.008,Y -147.290,Z 1522.913,A 0.000,B 0.000,C 90.000,E1 164.393} C_DIS
LIN {X 0.023,Y -150.608,Z 1522.888,A 0.000,B 0.000,C 90.000,E1 159.826} C_DIS
LIN {X -0.041,Y -154.083,Z 1522.868,A 0.000,B 0.000,C 90.000,E1 156.230} C_DIS
LIN {X 0.025,Y -157.503,Z 1522.848,A 0.000,B 0.000,C 90.000,E1 152.615} C_DIS
LIN {X -0.030,Y -161.734,Z 1522.828,A 0.000,B 0.000,C 90.000,E1 149.076} C_DIS
LIN {X -0.016,Y -165.927,Z 1522.809,A 0.000,B 0.000,C 90.000,E1 145.548} C_DIS
LIN {X -0.030,Y -170.915,Z 1522.789,A 0.000,B 0.000,C 90.000,E1 142.065} C_DIS
LIN {X -0.004,Y -175.783,Z 1522.770,A 0.000,B 0.000,C 90.000,E1 138.609} C_DIS
LIN {X -0.003,Y -181.391,Z 1522.751,A 0.000,B 0.000,C 90.000,E1 135.202} C_DIS
LIN {X 0.001,Y -186.889,Z 1522.732,A 0.000,B 0.000,C 90.000,E1 131.838} C_DIS
LIN {X -0.048,Y -191.471,Z 1522.719,A 0.000,B 0.000,C 90.000,E1 129.358} C_DIS
LIN {X -0.116,Y -197.330,Z 1522.700,A 0.000,B 0.000,C 90.000,E1 126.091} C_DIS
LIN {X 0.085,Y -200.607,Z 1522.691,A 0.000,B 0.000,C 90.000,E1 124.405} C_DIS
LIN {X 0.001,Y -202.446,Z 1522.685,A 0.000,B 0.000,C 90.000,E1 123.372} C_DIS
LIN {X -0.034,Y -317.214,Z 1522.685,A 0.000,B 0.000,C 90.000,E1 123.372} C_DIS
LIN {X 0.113,Y -319.674,Z 1522.685,A 0.000,B 0.000,C 90.000,E1 123.293} C_DIS
LIN {X -0.129,Y -324.246,Z 1522.684,A 0.000,B 0.000,C 90.000,E1 123.086} C_DIS
LIN {X -0.103,Y -326.902,Z 1522.682,A 0.000,B 0.000,C 90.000,E1 122.832} C_DIS
LIN {X -0.044,Y -330.613,Z 1522.679,A 0.000,B 0.000,C 90.000,E1 122.291} C_DIS
LIN {X 0.064,Y -332.148,Z 1522.678,A 0.000,B 0.000,C 90.000,E1 121.957} C_DIS
LIN {X -0.077,Y -344.583,Z 1522.660,A 0.000,B 0.000,C 90.000,E1 118.871} C_DIS
LIN {X 0.085,Y -357.193,Z 1522.645,A 0.000,B 0.000,C 90.000,E1 116.104} C_DIS
LIN {X -0.024,Y -371.303,Z 1522.630,A 0.000,B 0.000,C 90.000,E1 113.439} C_DIS
LIN {X 0.026,Y -385.209,Z 1522.617,A 0.000,B 0.000,C 90.000,E1 111.099} C_DIS
LIN {X -0.077,Y -400.497,Z 1522.605,A 0.000,B 0.000,C 90.000,E1 108.833} C_DIS
LIN {X -0.194,Y -417.272,Z 1522.592,A 0.000,B 0.000,C 90.000,E1 106.622} C_DIS
LIN {X 0.001,Y -435.652,Z 1522.580,A 0.000,B 0.000,C 90.000,E1 104.426} C_DIS
LIN {X -0.046,Y -455.416,Z 1522.569,A 0.000,B 0.000,C 90.000,E1 102.355} C_DIS
LIN {X 0.042,Y -475.785,Z 1522.558,A 0.000,B 0.000,C 90.000,E1 100.433} C_DIS
LIN {X 0.097,Y -491.336,Z 1522.551,A 0.000,B 0.000,C 90.000,E1 99.095} C_DIS
LIN {X -0.215,Y -493.352,Z 1522.549,A 0.000,B 0.000,C 90.000,E1 98.916} C_DIS
LIN {X 0.181,Y -495.088,Z 1522.548,A 0.000,B 0.000,C 90.000,E1 98.624} C_DIS
LIN {X 0.014,Y -496.386,Z 1522.547,A 0.000,B 0.000,C 90.000,E1 98.398} C_DIS
LIN {X -0.224,Y -497.979,Z 1522.544,A 0.000,B 0.000,C 90.000,E1 97.936} C_DIS
LIN {X 0.105,Y -498.490,Z 1522.541,A 0.000,B 0.000,C 90.000,E1 97.409} C_DIS
LIN {X -0.119,Y -498.004,Z 1522.539,A 0.000,B 0.000,C 90.000,E1 96.947} C_DIS
LIN {X 0.155,Y -496.449,Z 1522.536,A 0.000,B 0.000,C 90.000,E1 96.429} C_DIS
LIN {X 0.016,Y -495.185,Z 1522.534,A 0.000,B 0.000,C 90.000,E1 96.201} C_DIS
LIN {X 0.094,Y -483.858,Z 1522.525,A 0.000,B 0.000,C 90.000,E1 94.473} C_DIS
LIN {X 0.094,Y -474.665,Z 1522.517,A 0.000,B 0.000,C 90.000,E1 92.980} C_DIS
LIN {X 0.107,Y -466.496,Z 1522.510,A 0.000,B 0.000,C 90.000,E1 91.718} C_DIS
LIN {X -0.221,Y -456.197,Z 1522.501,A 0.000,B 0.000,C 90.000,E1 90.229} C_DIS
LIN {X 0.185,Y -445.496,Z 1522.493,A 0.000,B 0.000,C 90.000,E1 88.625} C_DIS
LIN {X -0.200,Y -436.321,Z 1522.485,A 0.000,B 0.000,C 90.000,E1 87.364} C_DIS
LIN {X 0.009,Y -423.236,Z 1522.475,A 0.000,B 0.000,C 90.000,E1 85.469} C_DIS
LIN {X 0.095,Y -408.491,Z 1522.463,A 0.000,B 0.000,C 90.000,E1 83.280} C_DIS
LIN {X -0.041,Y -391.985,Z 1522.449,A 0.000,B 0.000,C 90.000,E1 80.792} C_DIS
LIN {X -0.071,Y -372.979,Z 1522.431,A 0.000,B 0.000,C 90.000,E1 77.645} C_DIS
LIN {X 0.003,Y -359.899,Z 1522.418,A 0.000,B 0.000,C 90.000,E1 75.283} C_DIS
LIN {X -0.070,Y -348.643,Z 1522.407,A 0.000,B 0.000,C 90.000,E1 73.196} C_DIS
LIN {X 0.043,Y -337.437,Z 1522.395,A 0.000,B 0.000,C 90.000,E1 71.040} C_DIS
LIN {X 0.006,Y -322.186,Z 1522.377,A 0.000,B 0.000,C 90.000,E1 67.922} C_DIS
LIN {X -0.039,Y -309.024,Z 1522.361,A 0.000,B 0.000,C 90.000,E1 65.049} C_DIS
LIN {X 0.075,Y -297.826,Z 1522.347,A 0.000,B 0.000,C 90.000,E1 62.410} C_DIS
LIN {X 0.048,Y -286.908,Z 1522.332,A 0.000,B 0.000,C 90.000,E1 59.744} C_DIS
LIN {X -0.014,Y -277.617,Z 1522.319,A 0.000,B 0.000,C 90.000,E1 57.375} C_DIS
LIN {X -0.043,Y -267.167,Z 1522.303,A 0.000,B 0.000,C 90.000,E1 54.609} C_DIS
LIN {X -0.027,Y -257.108,Z 1522.288,A 0.000,B 0.000,C 90.000,E1 51.778} C_DIS
LIN {X -0.011,Y -246.325,Z 1522.270,A 0.000,B 0.000,C 90.000,E1 48.528} C_DIS
LIN {X 0.066,Y -237.523,Z 1522.253,A 0.000,B 0.000,C 90.000,E1 45.567} C_DIS
LIN {X -0.062,Y -229.460,Z 1522.237,A 0.000,B 0.000,C 90.000,E1 42.609} C_DIS
LIN {X -0.034,Y -222.162,Z 1522.220,A 0.000,B 0.000,C 90.000,E1 39.564} C_DIS
LIN {X 0.047,Y -215.637,Z 1522.203,A 0.000,B 0.000,C 90.000,E1 36.457} C_DIS
LIN {X -0.109,Y -209.843,Z 1522.185,A 0.000,B 0.000,C 90.000,E1 33.372} C_DIS
LIN {X -0.113,Y -203.488,Z 1522.163,A 0.000,B 0.000,C 90.000,E1 29.411} C_DIS
LIN {X 0.094,Y -197.917,Z 1522.141,A 0.000,B 0.000,C 90.000,E1 25.335} C_DIS
LIN {X 0.058,Y -193.187,Z 1522.118,A 0.000,B 0.000,C 90.000,E1 21.280} C_DIS
LIN {X -0.099,Y -189.289,Z 1522.095,A 0.000,B 0.000,C 90.000,E1 17.221} C_DIS
LIN {X -0.083,Y -185.446,Z 1522.068,A 0.000,B 0.000,C 90.000,E1 12.243} C_DIS
LIN {X -0.023,Y -182.324,Z 1522.035,A 0.000,B 0.000,C 90.000,E1 6.372} C_DIS
LIN {X -0.060,Y -180.687,Z 1521.983,A 0.000,B 0.000,C 90.000,E1 357.020} C_DIS
LIN {X -0.007,Y -182.534,Z 1521.937,A 0.000,B 0.000,C 90.000,E1 348.578} C_DIS
LIN {X -0.049,Y -185.294,Z 1521.909,A 0.000,B 0.000,C 90.000,E1 343.559} C_DIS
LIN {X 0.026,Y -189.203,Z 1521.881,A 0.000,B 0.000,C 90.000,E1 338.539} C_DIS
LIN {X 0.034,Y -193.477,Z 1521.858,A 0.000,B 0.000,C 90.000,E1 334.409} C_DIS
LIN {X -0.006,Y -198.662,Z 1521.835,A 0.000,B 0.000,C 90.000,E1 330.333} C_DIS
LIN {X -0.086,Y -203.525,Z 1521.817,A 0.000,B 0.000,C 90.000,E1 327.120} C_DIS
LIN {X -0.050,Y -209.078,Z 1521.799,A 0.000,B 0.000,C 90.000,E1 323.909} C_DIS
LIN {X 0.044,Y -215.405,Z 1521.782,A 0.000,B 0.000,C 90.000,E1 320.723} C_DIS
LIN {X -0.069,Y -222.552,Z 1521.765,A 0.000,B 0.000,C 90.000,E1 317.634} C_DIS
LIN {X -0.089,Y -231.571,Z 1521.745,A 0.000,B 0.000,C 90.000,E1 314.190} C_DIS
LIN {X 0.080,Y -239.545,Z 1521.731,A 0.000,B 0.000,C 90.000,E1 311.515} C_DIS
LIN {X -0.045,Y -247.323,Z 1521.718,A 0.000,B 0.000,C 90.000,E1 309.322} C_DIS
LIN {X -0.010,Y -254.540,Z 1521.708,A 0.000,B 0.000,C 90.000,E1 307.488} C_DIS
LIN {X 0.155,Y -261.029,Z 1521.700,A 0.000,B 0.000,C 90.000,E1 306.011} C_DIS
LIN {X -0.051,Y -270.211,Z 1521.690,A 0.000,B 0.000,C 90.000,E1 304.278} C_DIS
LIN {X -0.111,Y -280.531,Z 1521.681,A 0.000,B 0.000,C 90.000,E1 302.546} C_DIS
LIN {X 0.105,Y -289.506,Z 1521.673,A 0.000,B 0.000,C 90.000,E1 301.131} C_DIS
LIN {X -0.083,Y -306.605,Z 1521.660,A 0.000,B 0.000,C 90.000,E1 298.821} C_DIS
LIN {X 0.024,Y -330.427,Z 1521.644,A 0.000,B 0.000,C 90.000,E1 295.924} C_DIS
LIN {X -0.201,Y -349.069,Z 1521.633,A 0.000,B 0.000,C 90.000,E1 293.898} C_DIS
LIN {X 0.114,Y -365.207,Z 1521.623,A 0.000,B 0.000,C 90.000,E1 292.153} C_DIS
LIN {X -0.041,Y -378.375,Z 1521.615,A 0.000,B 0.000,C 90.000,E1 290.791} C_DIS
LIN {X 0.103,Y -386.003,Z 1521.611,A 0.000,B 0.000,C 90.000,E1 289.939} C_DIS
LIN {X 0.075,Y -393.606,Z 1521.606,A 0.000,B 0.000,C 90.000,E1 289.087} C_DIS
LIN {X 0.078,Y -400.707,Z 1521.601,A 0.000,B 0.000,C 90.000,E1 288.236} C_DIS
LIN {X 0.029,Y -407.188,Z 1521.597,A 0.000,B 0.000,C 90.000,E1 287.402} C_DIS
LIN {X 0.036,Y -413.068,Z 1521.592,A 0.000,B 0.000,C 90.000,E1 286.567} C_DIS
LIN {X 0.106,Y -418.222,Z 1521.588,A 0.000,B 0.000,C 90.000,E1 285.733} C_DIS
LIN {X 0.079,Y -421.222,Z 1521.584,A 0.000,B 0.000,C 90.000,E1 285.190} C_DIS
LIN {X 0.216,Y -425.001,Z 1521.580,A 0.000,B 0.000,C 90.000,E1 284.356} C_DIS
LIN {X 0.121,Y -427.160,Z 1521.577,A 0.000,B 0.000,C 90.000,E1 283.828} C_DIS
LIN {X 0.041,Y -428.975,Z 1521.574,A 0.000,B 0.000,C 90.000,E1 283.300} C_DIS
LIN {X -0.033,Y -430.391,Z 1521.571,A 0.000,B 0.000,C 90.000,E1 282.771} C_DIS
LIN {X -0.096,Y -431.464,Z 1521.568,A 0.000,B 0.000,C 90.000,E1 282.243} C_DIS
LIN {X -0.151,Y -432.006,Z 1521.565,A 0.000,B 0.000,C 90.000,E1 281.715} C_DIS
LIN {X -0.201,Y -432.129,Z 1521.562,A 0.000,B 0.000,C 90.000,E1 281.186} C_DIS
LIN {X 0.175,Y -431.683,Z 1521.559,A 0.000,B 0.000,C 90.000,E1 280.602} C_DIS
LIN {X 0.125,Y -430.640,Z 1521.556,A 0.000,B 0.000,C 90.000,E1 280.074} C_DIS
LIN {X -0.001,Y -429.044,Z 1521.553,A 0.000,B 0.000,C 90.000,E1 279.557} C_DIS
LIN {X -0.062,Y -426.758,Z 1521.550,A 0.000,B 0.000,C 90.000,E1 279.029} C_DIS
LIN {X -0.204,Y -423.695,Z 1521.547,A 0.000,B 0.000,C 90.000,E1 278.511} C_DIS
LIN {X 0.059,Y -419.765,Z 1521.544,A 0.000,B 0.000,C 90.000,E1 277.936} C_DIS
LIN {X -0.058,Y -414.814,Z 1521.541,A 0.000,B 0.000,C 90.000,E1 277.409} C_DIS
LIN {X -0.167,Y -408.900,Z 1521.538,A 0.000,B 0.000,C 90.000,E1 276.891} C_DIS
LIN {X 0.185,Y -402.861,Z 1521.536,A 0.000,B 0.000,C 90.000,E1 276.372} C_DIS
LIN {X 0.067,Y -396.651,Z 1521.533,A 0.000,B 0.000,C 90.000,E1 275.967} C_DIS
LIN {X -0.187,Y -390.248,Z 1521.531,A 0.000,B 0.000,C 90.000,E1 275.625} C_DIS
LIN {X -0.011,Y -380.644,Z 1521.528,A 0.000,B 0.000,C 90.000,E1 275.106} C_DIS
LIN {X 0.165,Y -370.729,Z 1521.526,A 0.000,B 0.000,C 90.000,E1 274.645} C_DIS
LIN {X 0.062,Y -352.064,Z 1521.522,A 0.000,B 0.000,C 90.000,E1 273.898} C_DIS
LIN {X -0.099,Y -342.253,Z 1521.520,A 0.000,B 0.000,C 90.000,E1 273.555} C_DIS
LIN {X 0.069,Y -328.942,Z 1521.517,A 0.000,B 0.000,C 90.000,E1 273.094} C_DIS
LIN {X -0.114,Y -315.418,Z 1521.515,A 0.000,B 0.000,C 90.000,E1 272.751} C_DIS
LIN {X 0.121,Y -304.016,Z 1521.514,A 0.000,B 0.000,C 90.000,E1 272.465} C_DIS
LIN {X 0.025,Y -291.665,Z 1521.513,A 0.000,B 0.000,C 90.000,E1 272.293} C_DIS
LIN {X -0.056,Y -278.219,Z 1521.512,A 0.000,B 0.000,C 90.000,E1 272.178} C_DIS
LIN {X 0.054,Y -268.440,Z 1521.512,A 0.000,B 0.000,C 90.000,E1 272.121} C_DIS
LIN {X 0.007,Y -181.242,Z 1521.512,A 0.000,B 0.000,C 90.000,E1 272.121} C_DIS
LIN {X -0.056,Y -181.577,Z 1521.502,A 0.000,B 0.000,C 90.000,E1 270.401} C_DIS
LIN {X -0.079,Y -180.906,Z 1521.474,A 0.000,B 0.000,C 90.000,E1 265.355} C_DIS
LIN {X -0.005,Y -180.669,Z 1521.469,A 0.000,B 0.000,C 90.000,E1 264.489} C_DIS
LIN {X 0.069,Y -178.750,Z 1521.441,A 0.000,B 0.000,C 90.000,E1 259.398} C_DIS
LIN {X -0.033,Y -175.797,Z 1521.413,A 0.000,B 0.000,C 90.000,E1 254.338} C_DIS
LIN {X -0.038,Y -171.983,Z 1521.384,A 0.000,B 0.000,C 90.000,E1 249.209} C_DIS
LIN {X -0.001,Y -171.388,Z 1521.380,A 0.000,B 0.000,C 90.000,E1 248.337} C_DIS
LIN {X -0.015,Y -167.632,Z 1521.356,A 0.000,B 0.000,C 90.000,E1 244.024} C_DIS
LIN {X 0.000,Y -166.289,Z 1521.346,A 0.000,B 0.000,C 90.000,E1 242.281} C_DIS
LIN {X -0.006,Y -163.036,Z 1521.327,A 0.000,B 0.000,C 90.000,E1 238.791} C_DIS
LIN {X -0.045,Y -160.966,Z 1521.312,A 0.000,B 0.000,C 90.000,E1 236.167} C_DIS
LIN {X -0.066,Y -157.719,Z 1521.292,A 0.000,B 0.000,C 90.000,E1 232.637} C_DIS
LIN {X 0.092,Y -155.758,Z 1521.277,A 0.000,B 0.000,C 90.000,E1 229.908} C_DIS
LIN {X -0.071,Y -152.014,Z 1521.253,A 0.000,B 0.000,C 90.000,E1 225.486} C_DIS
LIN {X -0.053,Y -150.261,Z 1521.238,A 0.000,B 0.000,C 90.000,E1 222.771} C_DIS
LIN {X -0.034,Y -147.015,Z 1521.212,A 0.000,B 0.000,C 90.000,E1 218.222} C_DIS
LIN {X -0.014,Y -145.598,Z 1521.197,A 0.000,B 0.000,C 90.000,E1 215.471} C_DIS
LIN {X -0.009,Y -142.984,Z 1521.172,A 0.000,B 0.000,C 90.000,E1 210.875} C_DIS
LIN {X -0.009,Y -141.612,Z 1521.151,A 0.000,B 0.000,C 90.000,E1 207.180} C_DIS
LIN {X 0.032,Y -139.428,Z 1521.115,A 0.000,B 0.000,C 90.000,E1 200.663} C_DIS
LIN {X 0.083,Y -139.157,Z 1521.104,A 0.000,B 0.000,C 90.000,E1 198.779} C_DIS
LIN {X -0.031,Y -138.343,Z 1521.058,A 0.000,B 0.000,C 90.000,E1 190.423} C_DIS
LIN {X -0.049,Y -139.481,Z 1521.006,A 0.000,B 0.000,C 90.000,E1 181.088} C_DIS
LIN {X 0.031,Y -141.073,Z 1520.975,A 0.000,B 0.000,C 90.000,E1 175.469} C_DIS
LIN {X -0.015,Y -142.449,Z 1520.959,A 0.000,B 0.000,C 90.000,E1 172.704} C_DIS
LIN {X 0.076,Y -144.690,Z 1520.934,A 0.000,B 0.000,C 90.000,E1 168.049} C_DIS
LIN {X 0.028,Y -147.283,Z 1520.913,A 0.000,B 0.000,C 90.000,E1 164.393} C_DIS
LIN {X 0.044,Y -150.601,Z 1520.888,A 0.000,B 0.000,C 90.000,E1 159.826} C_DIS
LIN {X -0.019,Y -154.074,Z 1520.868,A 0.000,B 0.000,C 90.000,E1 156.230} C_DIS
LIN {X 0.047,Y -157.495,Z 1520.848,A 0.000,B 0.000,C 90.000,E1 152.615} C_DIS
LIN {X -0.008,Y -161.723,Z 1520.828,A 0.000,B 0.000,C 90.000,E1 149.076} C_DIS
LIN {X 0.006,Y -165.916,Z 1520.809,A 0.000,B 0.000,C 90.000,E1 145.548} C_DIS
LIN {X -0.008,Y -170.902,Z 1520.789,A 0.000,B 0.000,C 90.000,E1 142.065} C_DIS
LIN {X 0.019,Y -175.771,Z 1520.770,A 0.000,B 0.000,C 90.000,E1 138.609} C_DIS
LIN {X 0.020,Y -181.380,Z 1520.751,A 0.000,B 0.000,C 90.000,E1 135.202} C_DIS
LIN {X 0.024,Y -186.877,Z 1520.732,A 0.000,B 0.000,C 90.000,E1 131.838} C_DIS
LIN {X -0.023,Y -191.460,Z 1520.719,A 0.000,B 0.000,C 90.000,E1 129.358} C_DIS
LIN {X -0.091,Y -197.316,Z 1520.700,A 0.000,B 0.000,C 90.000,E1 126.091} C_DIS
LIN {X 0.110,Y -200.592,Z 1520.691,A 0.000,B 0.000,C 90.000,E1 124.405} C_DIS
LIN {X -0.021,Y -202.373,Z 1520.686,A 0.000,B 0.000,C 90.000,E1 123.420} C_DIS
LIN {X -0.080,Y -316.174,Z 1520.686,A 0.000,B 0.000,C 90.000,E1 123.420} C_DIS
LIN {X 0.041,Y -318.327,Z 1520.685,A 0.000,B 0.000,C 90.000,E1 123.372} C_DIS
LIN {X 0.078,Y -324.066,Z 1520.684,A 0.000,B 0.000,C 90.000,E1 123.086} C_DIS
LIN {X -0.062,Y -326.995,Z 1520.682,A 0.000,B 0.000,C 90.000,E1 122.832} C_DIS
LIN {X -0.039,Y -330.645,Z 1520.679,A 0.000,B 0.000,C 90.000,E1 122.291} C_DIS
LIN {X 0.069,Y -332.140,Z 1520.678,A 0.000,B 0.000,C 90.000,E1 121.957} C_DIS
LIN {X -0.071,Y -344.558,Z 1520.660,A 0.000,B 0.000,C 90.000,E1 118.871} C_DIS
LIN {X 0.090,Y -357.166,Z 1520.645,A 0.000,B 0.000,C 90.000,E1 116.104} C_DIS
LIN {X -0.020,Y -371.276,Z 1520.630,A 0.000,B 0.000,C 90.000,E1 113.439} C_DIS
LIN {X 0.030,Y -385.182,Z 1520.617,A 0.000,B 0.000,C 90.000,E1 111.099} C_DIS
LIN {X -0.074,Y -400.469,Z 1520.605,A 0.000,B 0.000,C 90.000,E1 108.833} C_DIS
LIN {X -0.192,Y -417.242,Z 1520.592,A 0.000,B 0.000,C 90.000,E1 106.622} C_DIS
LIN {X 0.003,Y -435.622,Z 1520.580,A 0.000,B 0.000,C 90.000,E1 104.426} C_DIS
LIN {X -0.045,Y -455.386,Z 1520.569,A 0.000,B 0.000,C 90.000,E1 102.355} C_DIS
LIN {X 0.042,Y -475.754,Z 1520.558,A 0.000,B 0.000,C 90.000,E1 100.433} C_DIS
LIN {X 0.097,Y -491.298,Z 1520.551,A 0.000,B 0.000,C 90.000,E1 99.095} C_DIS
LIN {X -0.216,Y -493.299,Z 1520.549,A 0.000,B 0.000,C 90.000,E1 98.916} C_DIS
LIN {X 0.181,Y -495.023,Z 1520.548,A 0.000,B 0.000,C 90.000,E1 98.624} C_DIS
LIN {X 0.014,Y -496.311,Z 1520.547,A 0.000,B 0.000,C 90.000,E1 98.398} C_DIS
LIN {X -0.225,Y -497.892,Z 1520.544,A 0.000,B 0.000,C 90.000,E1 97.936} C_DIS
LIN {X 0.104,Y -498.391,Z 1520.541,A 0.000,B 0.000,C 90.000,E1 97.409} C_DIS
LIN {X -0.120,Y -497.895,Z 1520.539,A 0.000,B 0.000,C 90.000,E1 96.947} C_DIS
LIN {X 0.152,Y -496.327,Z 1520.536,A 0.000,B 0.000,C 90.000,E1 96.429} C_DIS
LIN {X 0.014,Y -495.055,Z 1520.534,A 0.000,B 0.000,C 90.000,E1 96.201} C_DIS
LIN {X 0.089,Y -483.716,Z 1520.525,A 0.000,B 0.000,C 90.000,E1 94.473} C_DIS
LIN {X 0.086,Y -474.533,Z 1520.517,A 0.000,B 0.000,C 90.000,E1 92.980} C_DIS
LIN {X 0.098,Y -466.381,Z 1520.510,A 0.000,B 0.000,C 90.000,E1 91.718} C_DIS
LIN {X 0.225,Y -456.086,Z 1520.501,A 0.000,B 0.000,C 90.000,E1 90.172} C_DIS
LIN {X -0.074,Y -443.608,Z 1520.491,A 0.000,B 0.000,C 90.000,E1 88.396} C_DIS
LIN {X -0.052,Y -434.390,Z 1520.484,A 0.000,B 0.000,C 90.000,E1 87.078} C_DIS
LIN {X -0.161,Y -419.529,Z 1520.472,A 0.000,B 0.000,C 90.000,E1 84.951} C_DIS
LIN {X -0.153,Y -404.801,Z 1520.460,A 0.000,B 0.000,C 90.000,E1 82.761} C_DIS
LIN {X 0.054,Y -386.666,Z 1520.444,A 0.000,B 0.000,C 90.000,E1 79.926} C_DIS
LIN {X 0.004,Y -368.047,Z 1520.426,A 0.000,B 0.000,C 90.000,E1 76.756} C_DIS
LIN {X -0.037,Y -355.063,Z 1520.413,A 0.000,B 0.000,C 90.000,E1 74.393} C_DIS
LIN {X 0.110,Y -343.836,Z 1520.401,A 0.000,B 0.000,C 90.000,E1 72.253} C_DIS
LIN {X -0.136,Y -329.678,Z 1520.386,A 0.000,B 0.000,C 90.000,E1 69.518} C_DIS
LIN {X -0.033,Y -317.708,Z 1520.372,A 0.000,B 0.000,C 90.000,E1 66.975} C_DIS
LIN {X -0.097,Y -306.169,Z 1520.358,A 0.000,B 0.000,C 90.000,E1 64.409} C_DIS
LIN {X -0.050,Y -295.073,Z 1520.343,A 0.000,B 0.000,C 90.000,E1 61.769} C_DIS
LIN {X -0.028,Y -282.952,Z 1520.326,A 0.000,B 0.000,C 90.000,E1 58.742} C_DIS
LIN {X -0.019,Y -273.757,Z 1520.313,A 0.000,B 0.000,C 90.000,E1 56.342} C_DIS
LIN {X -0.083,Y -262.242,Z 1520.296,A 0.000,B 0.000,C 90.000,E1 53.210} C_DIS
LIN {X -0.050,Y -251.206,Z 1520.278,A 0.000,B 0.000,C 90.000,E1 49.989} C_DIS
LIN {X -0.024,Y -242.035,Z 1520.261,A 0.000,B 0.000,C 90.000,E1 47.067} C_DIS
LIN {X -0.046,Y -233.608,Z 1520.245,A 0.000,B 0.000,C 90.000,E1 44.109} C_DIS
LIN {X 0.065,Y -225.959,Z 1520.228,A 0.000,B 0.000,C 90.000,E1 41.067} C_DIS
LIN {X 0.027,Y -219.093,Z 1520.211,A 0.000,B 0.000,C 90.000,E1 38.016} C_DIS
LIN {X 0.074,Y -212.932,Z 1520.194,A 0.000,B 0.000,C 90.000,E1 34.898} C_DIS
LIN {X -0.080,Y -206.215,Z 1520.172,A 0.000,B 0.000,C 90.000,E1 31.003} C_DIS
LIN {X -0.046,Y -200.326,Z 1520.150,A 0.000,B 0.000,C 90.000,E1 27.001} C_DIS
LIN {X -0.023,Y -195.258,Z 1520.127,A 0.000,B 0.000,C 90.000,E1 22.950} C_DIS
LIN {X 0.011,Y -191.006,Z 1520.105,A 0.000,B 0.000,C 90.000,E1 18.852} C_DIS
LIN {X 0.056,Y -186.899,Z 1520.077,A 0.000,B 0.000,C 90.000,E1 13.883} C_DIS
LIN {X -0.045,Y -183.750,Z 1520.049,A 0.000,B 0.000,C 90.000,E1 8.916} C_DIS
LIN {X 0.031,Y -181.328,Z 1520.012,A 0.000,B 0.000,C 90.000,E1 2.178} C_DIS
LIN {X 0.060,Y -181.066,Z 1519.974,A 0.000,B 0.000,C 90.000,E1 355.298} C_DIS
LIN {X -0.047,Y -183.143,Z 1519.932,A 0.000,B 0.000,C 90.000,E1 347.757} C_DIS
LIN {X -0.021,Y -186.098,Z 1519.904,A 0.000,B 0.000,C 90.000,E1 342.725} C_DIS
LIN {X 0.066,Y -189.414,Z 1519.881,A 0.000,B 0.000,C 90.000,E1 338.539} C_DIS
LIN {X 0.081,Y -193.671,Z 1519.858,A 0.000,B 0.000,C 90.000,E1 334.409} C_DIS
LIN {X 0.048,Y -198.821,Z 1519.835,A 0.000,B 0.000,C 90.000,E1 330.333} C_DIS
LIN {X -0.026,Y -203.676,Z 1519.817,A 0.000,B 0.000,C 90.000,E1 327.120} C_DIS
LIN {X 0.015,Y -209.214,Z 1519.800,A 0.000,B 0.000,C 90.000,E1 323.909} C_DIS
LIN {X 0.115,Y -215.536,Z 1519.782,A 0.000,B 0.000,C 90.000,E1 320.723} C_DIS
LIN {X 0.008,Y -222.664,Z 1519.765,A 0.000,B 0.000,C 90.000,E1 317.634} C_DIS
LIN {X -0.006,Y -231.697,Z 1519.745,A 0.000,B 0.000,C 90.000,E1 314.190} C_DIS
LIN {X 0.010,Y -239.673,Z 1519.731,A 0.000,B 0.000,C 90.000,E1 311.553} C_DIS
LIN {X 0.050,Y -248.780,Z 1519.716,A 0.000,B 0.000,C 90.000,E1 308.955} C_DIS
LIN {X -0.048,Y -256.145,Z 1519.706,A 0.000,B 0.000,C 90.000,E1 307.156} C_DIS
LIN {X -0.072,Y -262.793,Z 1519.698,A 0.000,B 0.000,C 90.000,E1 305.724} C_DIS
LIN {X 0.055,Y -270.145,Z 1519.691,A 0.000,B 0.000,C 90.000,E1 304.278} C_DIS
LIN {X -0.003,Y -280.425,Z 1519.681,A 0.000,B 0.000,C 90.000,E1 302.546} C_DIS
LIN {X 0.170,Y -294.065,Z 1519.669,A 0.000,B 0.000,C 90.000,E1 300.463} C_DIS
LIN {X 0.088,Y -311.582,Z 1519.656,A 0.000,B 0.000,C 90.000,E1 298.153} C_DIS
LIN {X -0.115,Y -332.920,Z 1519.642,A 0.000,B 0.000,C 90.000,E1 295.668} C_DIS
LIN {X 0.030,Y -348.860,Z 1519.633,A 0.000,B 0.000,C 90.000,E1 293.898} C_DIS
LIN {X -0.031,Y -365.125,Z 1519.623,A 0.000,B 0.000,C 90.000,E1 292.206} C_DIS
LIN {X 0.196,Y -378.274,Z 1519.616,A 0.000,B 0.000,C 90.000,E1 290.791} C_DIS
LIN {X -0.005,Y -388.504,Z 1519.609,A 0.000,B 0.000,C 90.000,E1 289.704} C_DIS
LIN {X 0.044,Y -395.893,Z 1519.605,A 0.000,B 0.000,C 90.000,E1 288.852} C_DIS
LIN {X 0.076,Y -402.847,Z 1519.600,A 0.000,B 0.000,C 90.000,E1 288.000} C_DIS
LIN {X 0.042,Y -409.162,Z 1519.595,A 0.000,B 0.000,C 90.000,E1 287.166} C_DIS
LIN {X 0.192,Y -414.892,Z 1519.591,A 0.000,B 0.000,C 90.000,E1 286.315} C_DIS
LIN {X -0.134,Y -419.864,Z 1519.586,A 0.000,B 0.000,C 90.000,E1 285.536} C_DIS
LIN {X -0.118,Y -423.997,Z 1519.582,A 0.000,B 0.000,C 90.000,E1 284.717} C_DIS
LIN {X 0.043,Y -427.390,Z 1519.577,A 0.000,B 0.000,C 90.000,E1 283.883} C_DIS
LIN {X -0.037,Y -429.212,Z 1519.574,A 0.000,B 0.000,C 90.000,E1 283.355} C_DIS
LIN {X -0.111,Y -430.742,Z 1519.571,A 0.000,B 0.000,C 90.000,E1 282.827} C_DIS
LIN {X -0.174,Y -431.861,Z 1519.568,A 0.000,B 0.000,C 90.000,E1 282.299} C_DIS
LIN {X 0.195,Y -432.501,Z 1519.565,A 0.000,B 0.000,C 90.000,E1 281.715} C_DIS
LIN {X 0.147,Y -432.656,Z 1519.562,A 0.000,B 0.000,C 90.000,E1 281.186} C_DIS
LIN {X 0.102,Y -432.256,Z 1519.559,A 0.000,B 0.000,C 90.000,E1 280.658} C_DIS
LIN {X -0.021,Y -431.335,Z 1519.556,A 0.000,B 0.000,C 90.000,E1 280.141} C_DIS
LIN {X -0.070,Y -429.782,Z 1519.553,A 0.000,B 0.000,C 90.000,E1 279.613} C_DIS
LIN {X -0.193,Y -427.599,Z 1519.550,A 0.000,B 0.000,C 90.000,E1 279.095} C_DIS
LIN {X 0.155,Y -424.630,Z 1519.547,A 0.000,B 0.000,C 90.000,E1 278.511} C_DIS
LIN {X 0.005,Y -420.817,Z 1519.544,A 0.000,B 0.000,C 90.000,E1 277.992} C_DIS
LIN {X -0.106,Y -415.937,Z 1519.541,A 0.000,B 0.000,C 90.000,E1 277.466} C_DIS
LIN {X 0.013,Y -413.228,Z 1519.540,A 0.000,B 0.000,C 90.000,E1 277.182} C_DIS
LIN {X 0.141,Y -407.366,Z 1519.537,A 0.000,B 0.000,C 90.000,E1 276.663} C_DIS
LIN {X -0.143,Y -401.333,Z 1519.535,A 0.000,B 0.000,C 90.000,E1 276.258} C_DIS
LIN {X -0.129,Y -395.029,Z 1519.532,A 0.000,B 0.000,C 90.000,E1 275.853} C_DIS
LIN {X 0.093,Y -388.572,Z 1519.530,A 0.000,B 0.000,C 90.000,E1 275.454} C_DIS
LIN {X 0.190,Y -381.991,Z 1519.529,A 0.000,B 0.000,C 90.000,E1 275.106} C_DIS
LIN {X -0.146,Y -368.857,Z 1519.525,A 0.000,B 0.000,C 90.000,E1 274.588} C_DIS
LIN {X 0.139,Y -350.126,Z 1519.521,A 0.000,B 0.000,C 90.000,E1 273.784} C_DIS
LIN {X 0.021,Y -340.012,Z 1519.519,A 0.000,B 0.000,C 90.000,E1 273.440} C_DIS
LIN {X -0.046,Y -326.941,Z 1519.517,A 0.000,B 0.000,C 90.000,E1 273.037} C_DIS
LIN {X -0.018,Y -316.604,Z 1519.515,A 0.000,B 0.000,C 90.000,E1 272.751} C_DIS
LIN {X 0.020,Y -309.455,Z 1519.514,A 0.000,B 0.000,C 90.000,E1 272.579} C_DIS
LIN {X 0.130,Y -297.795,Z 1519.513,A 0.000,B 0.000,C 90.000,E1 272.350} C_DIS
LIN {X -0.142,Y -283.758,Z 1519.512,A 0.000,B 0.000,C 90.000,E1 272.236} C_DIS
LIN {X 0.121,Y -273.843,Z 1519.512,A 0.000,B 0.000,C 90.000,E1 272.121} C_DIS
LIN {X 0.074,Y -269.305,Z 1519.512,A 0.000,B 0.000,C 90.000,E1 272.121} C_DIS
LIN {X 0.019,Y -181.242,Z 1519.512,A 0.000,B 0.000,C 90.000,E1 272.121} C_DIS
LIN {X -0.022,Y -181.576,Z 1519.502,A 0.000,B 0.000,C 90.000,E1 270.401} C_DIS
LIN {X -0.045,Y -180.906,Z 1519.474,A 0.000,B 0.000,C 90.000,E1 265.355} C_DIS
LIN {X 0.028,Y -180.674,Z 1519.469,A 0.000,B 0.000,C 90.000,E1 264.489} C_DIS
LIN {X -0.072,Y -178.757,Z 1519.441,A 0.000,B 0.000,C 90.000,E1 259.454} C_DIS
LIN {X 0.001,Y -175.803,Z 1519.413,A 0.000,B 0.000,C 90.000,E1 254.338} C_DIS
LIN {X -0.006,Y -171.989,Z 1519.385,A 0.000,B 0.000,C 90.000,E1 249.209} C_DIS
LIN {X 0.033,Y -171.399,Z 1519.380,A 0.000,B 0.000,C 90.000,E1 248.337} C_DIS
LIN {X 0.018,Y -167.640,Z 1519.356,A 0.000,B 0.000,C 90.000,E1 244.024} C_DIS
LIN {X 0.032,Y -166.300,Z 1519.346,A 0.000,B 0.000,C 90.000,E1 242.281} C_DIS
LIN {X 0.026,Y -163.046,Z 1519.327,A 0.000,B 0.000,C 90.000,E1 238.791} C_DIS
LIN {X -0.012,Y -160.978,Z 1519.312,A 0.000,B 0.000,C 90.000,E1 236.167} C_DIS
LIN {X -0.035,Y -157.728,Z 1519.292,A 0.000,B 0.000,C 90.000,E1 232.637} C_DIS
LIN {X -0.096,Y -155.768,Z 1519.277,A 0.000,B 0.000,C 90.000,E1 229.989} C_DIS
LIN {X -0.040,Y -152.022,Z 1519.253,A 0.000,B 0.000,C 90.000,E1 225.486} C_DIS
LIN {X -0.022,Y -150.269,Z 1519.238,A 0.000,B 0.000,C 90.000,E1 222.771} C_DIS
LIN {X -0.004,Y -147.022,Z 1519.212,A 0.000,B 0.000,C 90.000,E1 218.222} C_DIS
LIN {X 0.016,Y -145.604,Z 1519.197,A 0.000,B 0.000,C 90.000,E1 215.471} C_DIS
LIN {X 0.020,Y -142.990,Z 1519.172,A 0.000,B 0.000,C 90.000,E1 210.875} C_DIS
LIN {X 0.020,Y -141.617,Z 1519.151,A 0.000,B 0.000,C 90.000,E1 207.180} C_DIS
LIN {X 0.061,Y -139.430,Z 1519.115,A 0.000,B 0.000,C 90.000,E1 200.663} C_DIS
LIN {X -0.019,Y -139.160,Z 1519.105,A 0.000,B 0.000,C 90.000,E1 198.833} C_DIS
LIN {X -0.002,Y -138.342,Z 1519.058,A 0.000,B 0.000,C 90.000,E1 190.423} C_DIS
LIN {X -0.020,Y -139.480,Z 1519.006,A 0.000,B 0.000,C 90.000,E1 181.088} C_DIS
LIN {X 0.061,Y -141.069,Z 1518.975,A 0.000,B 0.000,C 90.000,E1 175.469} C_DIS
LIN {X 0.016,Y -142.443,Z 1518.959,A 0.000,B 0.000,C 90.000,E1 172.704} C_DIS
LIN {X -0.036,Y -144.683,Z 1518.934,A 0.000,B 0.000,C 90.000,E1 168.105} C_DIS
LIN {X 0.059,Y -147.273,Z 1518.913,A 0.000,B 0.000,C 90.000,E1 164.393} C_DIS
LIN {X -0.066,Y -150.592,Z 1518.888,A 0.000,B 0.000,C 90.000,E1 159.880} C_DIS
LIN {X 0.012,Y -154.064,Z 1518.868,A 0.000,B 0.000,C 90.000,E1 156.230} C_DIS
LIN {X 0.079,Y -157.483,Z 1518.848,A 0.000,B 0.000,C 90.000,E1 152.615} C_DIS
LIN {X 0.024,Y -161.708,Z 1518.828,A 0.000,B 0.000,C 90.000,E1 149.076} C_DIS
LIN {X 0.038,Y -165.901,Z 1518.809,A 0.000,B 0.000,C 90.000,E1 145.548} C_DIS
LIN {X 0.026,Y -170.885,Z 1518.789,A 0.000,B 0.000,C 90.000,E1 142.065} C_DIS
LIN {X 0.053,Y -175.754,Z 1518.770,A 0.000,B 0.000,C 90.000,E1 138.609} C_DIS
LIN {X -0.074,Y -181.364,Z 1518.751,A 0.000,B 0.000,C 90.000,E1 135.243} C_DIS
LIN {X 0.059,Y -186.857,Z 1518.733,A 0.000,B 0.000,C 90.000,E1 131.838} C_DIS
LIN {X 0.012,Y -191.442,Z 1518.719,A 0.000,B 0.000,C 90.000,E1 129.358} C_DIS
LIN {X -0.055,Y -197.295,Z 1518.700,A 0.000,B 0.000,C 90.000,E1 126.091} C_DIS
LIN {X -0.019,Y -200.573,Z 1518.691,A 0.000,B 0.000,C 90.000,E1 124.452} C_DIS
LIN {X -0.027,Y -202.320,Z 1518.686,A 0.000,B 0.000,C 90.000,E1 123.452} C_DIS
LIN {X -0.078,Y -316.451,Z 1518.686,A 0.000,B 0.000,C 90.000,E1 123.452} C_DIS
LIN {X 0.099,Y -319.087,Z 1518.686,A 0.000,B 0.000,C 90.000,E1 123.372} C_DIS
LIN {X 0.138,Y -324.215,Z 1518.684,A 0.000,B 0.000,C 90.000,E1 123.086} C_DIS
LIN {X -0.003,Y -327.050,Z 1518.682,A 0.000,B 0.000,C 90.000,E1 122.832} C_DIS
LIN {X -0.057,Y -330.693,Z 1518.679,A 0.000,B 0.000,C 90.000,E1 122.291} C_DIS
LIN {X 0.051,Y -332.145,Z 1518.678,A 0.000,B 0.000,C 90.000,E1 121.957} C_DIS
LIN {X -0.090,Y -344.549,Z 1518.660,A 0.000,B 0.000,C 90.000,E1 118.871} C_DIS
LIN {X 0.071,Y -357.159,Z 1518.645,A 0.000,B 0.000,C 90.000,E1 116.104} C_DIS
LIN {X -0.041,Y -371.270,Z 1518.630,A 0.000,B 0.000,C 90.000,E1 113.439} C_DIS
LIN {X 0.008,Y -385.178,Z 1518.617,A 0.000,B 0.000,C 90.000,E1 111.099} C_DIS
LIN {X -0.096,Y -400.466,Z 1518.604,A 0.000,B 0.000,C 90.000,E1 108.833} C_DIS
LIN {X -0.216,Y -417.243,Z 1518.592,A 0.000,B 0.000,C 90.000,E1 106.622} C_DIS
LIN {X -0.021,Y -435.624,Z 1518.580,A 0.000,B 0.000,C 90.000,E1 104.426} C_DIS
LIN {X -0.069,Y -455.388,Z 1518.569,A 0.000,B 0.000,C 90.000,E1 102.355} C_DIS
LIN {X 0.017,Y -475.758,Z 1518.558,A 0.000,B 0.000,C 90.000,E1 100.433} C_DIS
LIN {X 0.073,Y -491.289,Z 1518.551,A 0.000,B 0.000,C 90.000,E1 99.095} C_DIS
LIN {X -0.240,Y -493.268,Z 1518.549,A 0.000,B 0.000,C 90.000,E1 98.916} C_DIS
LIN {X 0.156,Y -494.975,Z 1518.548,A 0.000,B 0.000,C 90.000,E1 98.624} C_DIS
LIN {X -0.011,Y -496.251,Z 1518.547,A 0.000,B 0.000,C 90.000,E1 98.398} C_DIS
LIN {X -0.249,Y -497.813,Z 1518.544,A 0.000,B 0.000,C 90.000,E1 97.936} C_DIS
LIN {X 0.078,Y -498.295,Z 1518.541,A 0.000,B 0.000,C 90.000,E1 97.409} C_DIS
LIN {X -0.146,Y -497.782,Z 1518.538,A 0.000,B 0.000,C 90.000,E1 96.947} C_DIS
LIN {X 0.126,Y -496.195,Z 1518.536,A 0.000,B 0.000,C 90.000,E1 96.429} C_DIS
LIN {X -0.013,Y -494.911,Z 1518.534,A 0.000,B 0.000,C 90.000,E1 96.201} C_DIS
LIN {X 0.217,Y -485.084,Z 1518.526,A 0.000,B 0.000,C 90.000,E1 94.702} C_DIS
LIN {X 0.206,Y -475.942,Z 1518.518,A 0.000,B 0.000,C 90.000,E1 93.212} C_DIS
LIN {X -0.219,Y -467.924,Z 1518.511,A 0.000,B 0.000,C 90.000,E1 92.007} C_DIS
LIN {X -0.045,Y -457.696,Z 1518.503,A 0.000,B 0.000,C 90.000,E1 90.458} C_DIS
LIN {X -0.062,Y -447.073,Z 1518.494,A 0.000,B 0.000,C 90.000,E1 88.912} C_DIS
LIN {X 0.013,Y -438.011,Z 1518.487,A 0.000,B 0.000,C 90.000,E1 87.593} C_DIS
LIN {X -0.165,Y -425.003,Z 1518.476,A 0.000,B 0.000,C 90.000,E1 85.755} C_DIS
LIN {X -0.150,Y -412.112,Z 1518.466,A 0.000,B 0.000,C 90.000,E1 83.856} C_DIS
LIN {X -0.044,Y -401.095,Z 1518.457,A 0.000,B 0.000,C 90.000,E1 82.186} C_DIS
LIN {X 0.148,Y -381.466,Z 1518.439,A 0.000,B 0.000,C 90.000,E1 79.050} C_DIS
LIN {X -0.053,Y -364.765,Z 1518.423,A 0.000,B 0.000,C 90.000,E1 76.172} C_DIS
LIN {X -0.082,Y -351.828,Z 1518.410,A 0.000,B 0.000,C 90.000,E1 73.795} C_DIS
LIN {X 0.102,Y -340.657,Z 1518.398,A 0.000,B 0.000,C 90.000,E1 71.638} C_DIS
LIN {X 0.049,Y -325.131,Z 1518.381,A 0.000,B 0.000,C 90.000,E1 68.539} C_DIS
LIN {X 0.085,Y -311.871,Z 1518.365,A 0.000,B 0.000,C 90.000,E1 65.665} C_DIS
LIN {X 0.018,Y -299.189,Z 1518.349,A 0.000,B 0.000,C 90.000,E1 62.743} C_DIS
LIN {X 0.024,Y -288.284,Z 1518.334,A 0.000,B 0.000,C 90.000,E1 60.078} C_DIS
LIN {X -0.049,Y -277.748,Z 1518.319,A 0.000,B 0.000,C 90.000,E1 57.375} C_DIS
LIN {X -0.071,Y -267.417,Z 1518.303,A 0.000,B 0.000,C 90.000,E1 54.609} C_DIS
LIN {X -0.049,Y -257.387,Z 1518.288,A 0.000,B 0.000,C 90.000,E1 51.778} C_DIS
LIN {X -0.023,Y -246.696,Z 1518.270,A 0.000,B 0.000,C 90.000,E1 48.528} C_DIS
LIN {X 0.065,Y -237.950,Z 1518.253,A 0.000,B 0.000,C 90.000,E1 45.567} C_DIS
LIN {X -0.053,Y -229.919,Z 1518.237,A 0.000,B 0.000,C 90.000,E1 42.609} C_DIS
LIN {X -0.015,Y -222.660,Z 1518.220,A 0.000,B 0.000,C 90.000,E1 39.564} C_DIS
LIN {X -0.095,Y -216.193,Z 1518.203,A 0.000,B 0.000,C 90.000,E1 36.503} C_DIS
LIN {X -0.066,Y -210.428,Z 1518.185,A 0.000,B 0.000,C 90.000,E1 33.372} C_DIS
LIN {X -0.052,Y -204.064,Z 1518.163,A 0.000,B 0.000,C 90.000,E1 29.411} C_DIS
LIN {X -0.094,Y -198.479,Z 1518.141,A 0.000,B 0.000,C 90.000,E1 25.412} C_DIS
LIN {X -0.030,Y -193.721,Z 1518.119,A 0.000,B 0.000,C 90.000,E1 21.334} C_DIS
LIN {X 0.007,Y -189.811,Z 1518.096,A 0.000,B 0.000,C 90.000,E1 17.221} C_DIS
LIN {X 0.041,Y -185.970,Z 1518.068,A 0.000,B 0.000,C 90.000,E1 12.243} C_DIS
LIN {X -0.061,Y -182.855,Z 1518.036,A 0.000,B 0.000,C 90.000,E1 6.429} C_DIS
LIN {X -0.050,Y -181.220,Z 1517.983,A 0.000,B 0.000,C 90.000,E1 357.020} C_DIS
LIN {X 0.035,Y -183.026,Z 1517.937,A 0.000,B 0.000,C 90.000,E1 348.578} C_DIS
LIN {X 0.013,Y -185.760,Z 1517.909,A 0.000,B 0.000,C 90.000,E1 343.559} C_DIS
LIN {X -0.071,Y -189.623,Z 1517.881,A 0.000,B 0.000,C 90.000,E1 338.592} C_DIS
LIN {X -0.048,Y -193.869,Z 1517.858,A 0.000,B 0.000,C 90.000,E1 334.460} C_DIS
LIN {X 0.102,Y -198.983,Z 1517.835,A 0.000,B 0.000,C 90.000,E1 330.333} C_DIS
LIN {X 0.033,Y -203.835,Z 1517.817,A 0.000,B 0.000,C 90.000,E1 327.120} C_DIS
LIN {X 0.081,Y -209.349,Z 1517.800,A 0.000,B 0.000,C 90.000,E1 323.909} C_DIS
LIN {X -0.118,Y -215.666,Z 1517.782,A 0.000,B 0.000,C 90.000,E1 320.803} C_DIS
LIN {X 0.083,Y -222.775,Z 1517.765,A 0.000,B 0.000,C 90.000,E1 317.634} C_DIS
LIN {X 0.076,Y -231.827,Z 1517.746,A 0.000,B 0.000,C 90.000,E1 314.190} C_DIS
LIN {X -0.105,Y -241.027,Z 1517.729,A 0.000,B 0.000,C 90.000,E1 311.229} C_DIS
LIN {X -0.011,Y -250.272,Z 1517.715,A 0.000,B 0.000,C 90.000,E1 308.624} C_DIS
LIN {X 0.080,Y -257.785,Z 1517.704,A 0.000,B 0.000,C 90.000,E1 306.790} C_DIS
LIN {X -0.075,Y -264.565,Z 1517.697,A 0.000,B 0.000,C 90.000,E1 305.391} C_DIS
LIN {X -0.148,Y -272.063,Z 1517.689,A 0.000,B 0.000,C 90.000,E1 303.992} C_DIS
LIN {X 0.048,Y -282.519,Z 1517.679,A 0.000,B 0.000,C 90.000,E1 302.212} C_DIS
LIN {X -0.120,Y -293.907,Z 1517.670,A 0.000,B 0.000,C 90.000,E1 300.541} C_DIS
LIN {X 0.173,Y -308.799,Z 1517.658,A 0.000,B 0.000,C 90.000,E1 298.487} C_DIS
LIN {X -0.086,Y -332.927,Z 1517.643,A 0.000,B 0.000,C 90.000,E1 295.668} C_DIS
LIN {X -0.004,Y -349.051,Z 1517.633,A 0.000,B 0.000,C 90.000,E1 293.898} C_DIS
LIN {X -0.030,Y -365.316,Z 1517.623,A 0.000,B 0.000,C 90.000,E1 292.206} C_DIS
LIN {X -0.108,Y -378.427,Z 1517.616,A 0.000,B 0.000,C 90.000,E1 290.844} C_DIS
LIN {X 0.046,Y -388.660,Z 1517.609,A 0.000,B 0.000,C 90.000,E1 289.704} C_DIS
LIN {X 0.075,Y -396.089,Z 1517.605,A 0.000,B 0.000,C 90.000,E1 288.852} C_DIS
LIN {X 0.110,Y -403.041,Z 1517.600,A 0.000,B 0.000,C 90.000,E1 288.000} C_DIS
LIN {X 0.078,Y -409.407,Z 1517.595,A 0.000,B 0.000,C 90.000,E1 287.166} C_DIS
LIN {X 0.232,Y -415.153,Z 1517.591,A 0.000,B 0.000,C 90.000,E1 286.315} C_DIS
LIN {X -0.091,Y -420.168,Z 1517.586,A 0.000,B 0.000,C 90.000,E1 285.536} C_DIS
LIN {X -0.072,Y -424.342,Z 1517.582,A 0.000,B 0.000,C 90.000,E1 284.717} C_DIS
LIN {X 0.092,Y -427.728,Z 1517.577,A 0.000,B 0.000,C 90.000,E1 283.883} C_DIS
LIN {X 0.014,Y -429.658,Z 1517.574,A 0.000,B 0.000,C 90.000,E1 283.355} C_DIS
LIN {X -0.058,Y -431.163,Z 1517.571,A 0.000,B 0.000,C 90.000,E1 282.827} C_DIS
LIN {X -0.118,Y -432.323,Z 1517.568,A 0.000,B 0.000,C 90.000,E1 282.299} C_DIS
LIN {X -0.170,Y -432.997,Z 1517.565,A 0.000,B 0.000,C 90.000,E1 281.771} C_DIS
LIN {X 0.209,Y -433.177,Z 1517.562,A 0.000,B 0.000,C 90.000,E1 281.186} C_DIS
LIN {X 0.166,Y -432.819,Z 1517.559,A 0.000,B 0.000,C 90.000,E1 280.658} C_DIS
LIN {X 0.046,Y -431.925,Z 1517.556,A 0.000,B 0.000,C 90.000,E1 280.141} C_DIS
LIN {X 0.001,Y -430.407,Z 1517.553,A 0.000,B 0.000,C 90.000,E1 279.613} C_DIS
LIN {X -0.121,Y -428.253,Z 1517.550,A 0.000,B 0.000,C 90.000,E1 279.095} C_DIS
LIN {X -0.182,Y -425.333,Z 1517.547,A 0.000,B 0.000,C 90.000,E1 278.568} C_DIS
LIN {X 0.090,Y -421.529,Z 1517.544,A 0.000,B 0.000,C 90.000,E1 277.992} C_DIS
LIN {X -0.018,Y -416.758,Z 1517.542,A 0.000,B 0.000,C 90.000,E1 277.466} C_DIS
LIN {X 0.086,Y -414.016,Z 1517.540,A 0.000,B 0.000,C 90.000,E1 277.182} C_DIS
LIN {X 0.181,Y -408.135,Z 1517.537,A 0.000,B 0.000,C 90.000,E1 276.663} C_DIS
LIN {X -0.134,Y -402.029,Z 1517.535,A 0.000,B 0.000,C 90.000,E1 276.258} C_DIS
LIN {X -0.139,Y -395.722,Z 1517.532,A 0.000,B 0.000,C 90.000,E1 275.853} C_DIS
LIN {X 0.099,Y -389.292,Z 1517.530,A 0.000,B 0.000,C 90.000,E1 275.454} C_DIS
LIN {X -0.157,Y -382.791,Z 1517.529,A 0.000,B 0.000,C 90.000,E1 275.163} C_DIS
LIN {X 0.013,Y -372.884,Z 1517.526,A 0.000,B 0.000,C 90.000,E1 274.702} C_DIS
LIN {X -0.091,Y -357.070,Z 1517.523,A 0.000,B 0.000,C 90.000,E1 274.073} C_DIS
LIN {X 0.105,Y -347.463,Z 1517.521,A 0.000,B 0.000,C 90.000,E1 273.669} C_DIS
LIN {X 0.133,Y -337.651,Z 1517.519,A 0.000,B 0.000,C 90.000,E1 273.326} C_DIS
LIN {X 0.012,Y -327.826,Z 1517.517,A 0.000,B 0.000,C 90.000,E1 273.037} C_DIS
LIN {X 0.044,Y -317.622,Z 1517.515,A 0.000,B 0.000,C 90.000,E1 272.751} C_DIS
LIN {X -0.052,Y -306.284,Z 1517.514,A 0.000,B 0.000,C 90.000,E1 272.522} C_DIS
LIN {X 0.147,Y -298.640,Z 1517.513,A 0.000,B 0.000,C 90.000,E1 272.350} C_DIS
LIN {X -0.140,Y -284.336,Z 1517.512,A 0.000,B 0.000,C 90.000,E1 272.236} C_DIS
LIN {X -0.100,Y -276.673,Z 1517.512,A 0.000,B 0.000,C 90.000,E1 272.178} C_DIS
LIN {X 0.082,Y -270.718,Z 1517.512,A 0.000,B 0.000,C 90.000,E1 272.121} C_DIS
LIN {X 0.025,Y -181.241,Z 1517.512,A 0.000,B 0.000,C 90.000,E1 272.121} C_DIS
LIN {X -0.014,Y -181.576,Z 1517.502,A 0.000,B 0.000,C 90.000,E1 270.401} C_DIS
LIN {X -0.037,Y -180.905,Z 1517.474,A 0.000,B 0.000,C 90.000,E1 265.355} C_DIS
LIN {X 0.037,Y -180.676,Z 1517.469,A 0.000,B 0.000,C 90.000,E1 264.489} C_DIS
LIN {X -0.065,Y -178.758,Z 1517.441,A 0.000,B 0.000,C 90.000,E1 259.454} C_DIS
LIN {X 0.007,Y -175.805,Z 1517.413,A 0.000,B 0.000,C 90.000,E1 254.338} C_DIS
LIN {X 0.002,Y -171.991,Z 1517.385,A 0.000,B 0.000,C 90.000,E1 249.209} C_DIS
LIN {X 0.040,Y -171.400,Z 1517.380,A 0.000,B 0.000,C 90.000,E1 248.337} C_DIS
LIN {X 0.025,Y -167.642,Z 1517.356,A 0.000,B 0.000,C 90.000,E1 244.024} C_DIS
LIN {X 0.040,Y -166.303,Z 1517.346,A 0.000,B 0.000,C 90.000,E1 242.281} C_DIS
LIN {X 0.033,Y -163.047,Z 1517.327,A 0.000,B 0.000,C 90.000,E1 238.791} C_DIS
LIN {X -0.005,Y -160.981,Z 1517.312,A 0.000,B 0.000,C 90.000,E1 236.167} C_DIS
LIN {X -0.028,Y -157.730,Z 1517.292,A 0.000,B 0.000,C 90.000,E1 232.637} C_DIS
LIN {X -0.088,Y -155.769,Z 1517.278,A 0.000,B 0.000,C 90.000,E1 229.989} C_DIS
LIN {X -0.034,Y -152.024,Z 1517.253,A 0.000,B 0.000,C 90.000,E1 225.486} C_DIS
LIN {X -0.015,Y -150.272,Z 1517.238,A 0.000,B 0.000,C 90.000,E1 222.771} C_DIS
LIN {X 0.002,Y -147.024,Z 1517.212,A 0.000,B 0.000,C 90.000,E1 218.222} C_DIS
LIN {X 0.024,Y -145.606,Z 1517.197,A 0.000,B 0.000,C 90.000,E1 215.471} C_DIS
LIN {X 0.027,Y -142.992,Z 1517.172,A 0.000,B 0.000,C 90.000,E1 210.875} C_DIS
LIN {X -0.038,Y -141.618,Z 1517.151,A 0.000,B 0.000,C 90.000,E1 207.206} C_DIS
LIN {X 0.019,Y -139.430,Z 1517.115,A 0.000,B 0.000,C 90.000,E1 200.684} C_DIS
LIN {X -0.058,Y -139.160,Z 1517.105,A 0.000,B 0.000,C 90.000,E1 198.852} C_DIS
LIN {X -0.020,Y -138.342,Z 1517.058,A 0.000,B 0.000,C 90.000,E1 190.433} C_DIS
LIN {X -0.013,Y -139.480,Z 1517.006,A 0.000,B 0.000,C 90.000,E1 181.088} C_DIS
LIN {X 0.068,Y -141.067,Z 1516.975,A 0.000,B 0.000,C 90.000,E1 175.469} C_DIS
LIN {X 0.022,Y -142.442,Z 1516.959,A 0.000,B 0.000,C 90.000,E1 172.704} C_DIS
LIN {X -0.029,Y -144.682,Z 1516.934,A 0.000,B 0.000,C 90.000,E1 168.105} C_DIS
LIN {X 0.066,Y -147.271,Z 1516.913,A 0.000,B 0.000,C 90.000,E1 164.393} C_DIS
LIN {X -0.059,Y -150.589,Z 1516.888,A 0.000,B 0.000,C 90.000,E1 159.880} C_DIS
LIN {X 0.018,Y -154.061,Z 1516.868,A 0.000,B 0.000,C 90.000,E1 156.230} C_DIS
LIN {X -0.055,Y -157.480,Z 1516.848,A 0.000,B 0.000,C 90.000,E1 152.666} C_DIS
LIN {X 0.032,Y -161.705,Z 1516.828,A 0.000,B 0.000,C 90.000,E1 149.076} C_DIS
LIN {X -0.091,Y -165.899,Z 1516.809,A 0.000,B 0.000,C 90.000,E1 145.595} C_DIS
LIN {X 0.033,Y -170.882,Z 1516.789,A 0.000,B 0.000,C 90.000,E1 142.065} C_DIS
LIN {X 0.061,Y -175.750,Z 1516.770,A 0.000,B 0.000,C 90.000,E1 138.609} C_DIS
LIN {X -0.066,Y -181.361,Z 1516.751,A 0.000,B 0.000,C 90.000,E1 135.243} C_DIS
LIN {X 0.067,Y -186.852,Z 1516.733,A 0.000,B 0.000,C 90.000,E1 131.838} C_DIS
LIN {X 0.020,Y -191.438,Z 1516.719,A 0.000,B 0.000,C 90.000,E1 129.358} C_DIS
LIN {X -0.046,Y -197.290,Z 1516.700,A 0.000,B 0.000,C 90.000,E1 126.091} C_DIS
LIN {X -0.011,Y -200.568,Z 1516.691,A 0.000,B 0.000,C 90.000,E1 124.452} C_DIS
LIN {X -0.071,Y -202.258,Z 1516.686,A 0.000,B 0.000,C 90.000,E1 123.499} C_DIS
LIN {X -0.159,Y -316.379,Z 1516.686,A 0.000,B 0.000,C 90.000,E1 123.499} C_DIS
LIN {X 0.006,Y -317.755,Z 1516.686,A 0.000,B 0.000,C 90.000,E1 123.452} C_DIS
LIN {X 0.029,Y -321.844,Z 1516.685,A 0.000,B 0.000,C 90.000,E1 123.293} C_DIS
LIN {X -0.127,Y -324.088,Z 1516.684,A 0.000,B 0.000,C 90.000,E1 123.166} C_DIS
LIN {X 0.011,Y -327.167,Z 1516.682,A 0.000,B 0.000,C 90.000,E1 122.832} C_DIS
LIN {X -0.091,Y -330.750,Z 1516.679,A 0.000,B 0.000,C 90.000,E1 122.291} C_DIS
LIN {X -0.157,Y -333.340,Z 1516.676,A 0.000,B 0.000,C 90.000,E1 121.671} C_DIS
LIN {X -0.125,Y -344.552,Z 1516.660,A 0.000,B 0.000,C 90.000,E1 118.871} C_DIS
LIN {X 0.034,Y -357.165,Z 1516.645,A 0.000,B 0.000,C 90.000,E1 116.104} C_DIS
LIN {X -0.078,Y -371.279,Z 1516.630,A 0.000,B 0.000,C 90.000,E1 113.439} C_DIS
LIN {X -0.030,Y -385.189,Z 1516.617,A 0.000,B 0.000,C 90.000,E1 111.099} C_DIS
LIN {X 0.243,Y -400.481,Z 1516.604,A 0.000,B 0.000,C 90.000,E1 108.779} C_DIS
LIN {X 0.144,Y -417.261,Z 1516.592,A 0.000,B 0.000,C 90.000,E1 106.567} C_DIS
LIN {X 0.045,Y -435.646,Z 1516.580,A 0.000,B 0.000,C 90.000,E1 104.411} C_DIS
LIN {X -0.111,Y -455.413,Z 1516.569,A 0.000,B 0.000,C 90.000,E1 102.355} C_DIS
LIN {X -0.024,Y -475.784,Z 1516.558,A 0.000,B 0.000,C 90.000,E1 100.433} C_DIS
LIN {X 0.033,Y -491.298,Z 1516.551,A 0.000,B 0.000,C 90.000,E1 99.095} C_DIS
LIN {X 0.207,Y -493.248,Z 1516.549,A 0.000,B 0.000,C 90.000,E1 98.859} C_DIS
LIN {X 0.115,Y -494.932,Z 1516.548,A 0.000,B 0.000,C 90.000,E1 98.624} C_DIS
LIN {X -0.052,Y -496.191,Z 1516.547,A 0.000,B 0.000,C 90.000,E1 98.398} C_DIS
LIN {X 0.271,Y -497.726,Z 1516.544,A 0.000,B 0.000,C 90.000,E1 97.871} C_DIS
LIN {X 0.037,Y -498.187,Z 1516.541,A 0.000,B 0.000,C 90.000,E1 97.409} C_DIS
LIN {X -0.188,Y -497.654,Z 1516.538,A 0.000,B 0.000,C 90.000,E1 96.947} C_DIS
LIN {X 0.084,Y -496.042,Z 1516.536,A 0.000,B 0.000,C 90.000,E1 96.429} C_DIS
LIN {X -0.055,Y -494.741,Z 1516.534,A 0.000,B 0.000,C 90.000,E1 96.201} C_DIS
LIN {X 0.173,Y -484.907,Z 1516.526,A 0.000,B 0.000,C 90.000,E1 94.702} C_DIS
LIN {X 0.159,Y -475.793,Z 1516.518,A 0.000,B 0.000,C 90.000,E1 93.212} C_DIS
LIN {X 0.200,Y -467.769,Z 1516.511,A 0.000,B 0.000,C 90.000,E1 91.949} C_DIS
LIN {X -0.094,Y -457.548,Z 1516.502,A 0.000,B 0.000,C 90.000,E1 90.458} C_DIS
LIN {X -0.113,Y -446.940,Z 1516.494,A 0.000,B 0.000,C 90.000,E1 88.912} C_DIS
LIN {X -0.039,Y -437.920,Z 1516.487,A 0.000,B 0.000,C 90.000,E1 87.593} C_DIS
LIN {X 0.207,Y -424.939,Z 1516.476,A 0.000,B 0.000,C 90.000,E1 85.698} C_DIS
LIN {X 0.208,Y -412.075,Z 1516.466,A 0.000,B 0.000,C 90.000,E1 83.799} C_DIS
LIN {X -0.095,Y -401.086,Z 1516.457,A 0.000,B 0.000,C 90.000,E1 82.186} C_DIS
LIN {X 0.098,Y -381.463,Z 1516.439,A 0.000,B 0.000,C 90.000,E1 79.050} C_DIS
LIN {X -0.100,Y -364.755,Z 1516.423,A 0.000,B 0.000,C 90.000,E1 76.172} C_DIS
LIN {X -0.170,Y -353.432,Z 1516.411,A 0.000,B 0.000,C 90.000,E1 74.102} C_DIS
LIN {X 0.058,Y -340.651,Z 1516.398,A 0.000,B 0.000,C 90.000,E1 71.638} C_DIS
LIN {X 0.006,Y -325.102,Z 1516.381,A 0.000,B 0.000,C 90.000,E1 68.539} C_DIS
LIN {X 0.043,Y -311.842,Z 1516.365,A 0.000,B 0.000,C 90.000,E1 65.665} C_DIS
LIN {X -0.023,Y -299.162,Z 1516.349,A 0.000,B 0.000,C 90.000,E1 62.743} C_DIS
LIN {X -0.015,Y -288.284,Z 1516.334,A 0.000,B 0.000,C 90.000,E1 60.078} C_DIS
LIN {X -0.129,Y -276.502,Z 1516.317,A 0.000,B 0.000,C 90.000,E1 57.041} C_DIS
LIN {X -0.113,Y -265.000,Z 1516.299,A 0.000,B 0.000,C 90.000,E1 53.909} C_DIS
LIN {X 0.040,Y -253.894,Z 1516.282,A 0.000,B 0.000,C 90.000,E1 50.678} C_DIS
LIN {X 0.124,Y -243.536,Z 1516.263,A 0.000,B 0.000,C 90.000,E1 47.391} C_DIS
LIN {X -0.071,Y -234.051,Z 1516.245,A 0.000,B 0.000,C 90.000,E1 44.109} C_DIS
LIN {X 0.052,Y -226.430,Z 1516.228,A 0.000,B 0.000,C 90.000,E1 41.067} C_DIS
LIN {X 0.028,Y -219.607,Z 1516.211,A 0.000,B 0.000,C 90.000,E1 38.016} C_DIS
LIN {X 0.087,Y -213.503,Z 1516.194,A 0.000,B 0.000,C 90.000,E1 34.898} C_DIS
LIN {X -0.051,Y -206.811,Z 1516.172,A 0.000,B 0.000,C 90.000,E1 31.003} C_DIS
LIN {X 0.000,Y -200.868,Z 1516.150,A 0.000,B 0.000,C 90.000,E1 27.001} C_DIS
LIN {X 0.038,Y -195.801,Z 1516.128,A 0.000,B 0.000,C 90.000,E1 22.950} C_DIS
LIN {X -0.093,Y -191.529,Z 1516.105,A 0.000,B 0.000,C 90.000,E1 18.906} C_DIS
LIN {X -0.032,Y -187.398,Z 1516.077,A 0.000,B 0.000,C 90.000,E1 13.939} C_DIS
LIN {X 0.065,Y -184.261,Z 1516.050,A 0.000,B 0.000,C 90.000,E1 8.916} C_DIS
LIN {X -0.016,Y -181.864,Z 1516.012,A 0.000,B 0.000,C 90.000,E1 2.236} C_DIS
LIN {X 0.076,Y -181.604,Z 1515.974,A 0.000,B 0.000,C 90.000,E1 355.298} C_DIS
LIN {X -0.003,Y -183.626,Z 1515.932,A 0.000,B 0.000,C 90.000,E1 347.757} C_DIS
LIN {X 0.042,Y -186.552,Z 1515.904,A 0.000,B 0.000,C 90.000,E1 342.725} C_DIS
LIN {X -0.033,Y -189.822,Z 1515.881,A 0.000,B 0.000,C 90.000,E1 338.592} C_DIS
LIN {X -0.002,Y -194.046,Z 1515.858,A 0.000,B 0.000,C 90.000,E1 334.460} C_DIS
LIN {X -0.019,Y -199.148,Z 1515.835,A 0.000,B 0.000,C 90.000,E1 330.383} C_DIS
LIN {X 0.091,Y -203.981,Z 1515.818,A 0.000,B 0.000,C 90.000,E1 327.120} C_DIS
LIN {X 0.143,Y -209.491,Z 1515.800,A 0.000,B 0.000,C 90.000,E1 323.909} C_DIS
LIN {X -0.050,Y -215.792,Z 1515.782,A 0.000,B 0.000,C 90.000,E1 320.803} C_DIS
LIN {X -0.007,Y -222.891,Z 1515.765,A 0.000,B 0.000,C 90.000,E1 317.676} C_DIS
LIN {X -0.009,Y -231.965,Z 1515.746,A 0.000,B 0.000,C 90.000,E1 314.231} C_DIS
LIN {X -0.017,Y -241.173,Z 1515.729,A 0.000,B 0.000,C 90.000,E1 311.229} C_DIS
LIN {X 0.084,Y -250.377,Z 1515.715,A 0.000,B 0.000,C 90.000,E1 308.624} C_DIS
LIN {X 0.148,Y -256.273,Z 1515.707,A 0.000,B 0.000,C 90.000,E1 307.156} C_DIS
LIN {X 0.131,Y -262.850,Z 1515.699,A 0.000,B 0.000,C 90.000,E1 305.724} C_DIS
LIN {X 0.041,Y -270.099,Z 1515.691,A 0.000,B 0.000,C 90.000,E1 304.326} C_DIS
LIN {X -0.024,Y -280.251,Z 1515.681,A 0.000,B 0.000,C 90.000,E1 302.594} C_DIS
LIN {X -0.008,Y -293.761,Z 1515.670,A 0.000,B 0.000,C 90.000,E1 300.541} C_DIS
LIN {X -0.131,Y -308.608,Z 1515.659,A 0.000,B 0.000,C 90.000,E1 298.565} C_DIS
LIN {X 0.064,Y -332.753,Z 1515.643,A 0.000,B 0.000,C 90.000,E1 295.668} C_DIS
LIN {X 0.033,Y -349.146,Z 1515.633,A 0.000,B 0.000,C 90.000,E1 293.898} C_DIS
LIN {X -0.031,Y -364.988,Z 1515.624,A 0.000,B 0.000,C 90.000,E1 292.259} C_DIS
LIN {X 0.058,Y -378.196,Z 1515.616,A 0.000,B 0.000,C 90.000,E1 290.865} C_DIS
LIN {X 0.038,Y -388.413,Z 1515.610,A 0.000,B 0.000,C 90.000,E1 289.758} C_DIS
LIN {X 0.090,Y -395.823,Z 1515.605,A 0.000,B 0.000,C 90.000,E1 288.906} C_DIS
LIN {X 0.121,Y -402.845,Z 1515.600,A 0.000,B 0.000,C 90.000,E1 288.055} C_DIS
LIN {X 0.086,Y -409.299,Z 1515.596,A 0.000,B 0.000,C 90.000,E1 287.221} C_DIS
LIN {X 0.119,Y -415.111,Z 1515.591,A 0.000,B 0.000,C 90.000,E1 286.386} C_DIS
LIN {X 0.075,Y -418.596,Z 1515.588,A 0.000,B 0.000,C 90.000,E1 285.843} C_DIS
LIN {X 0.188,Y -423.094,Z 1515.583,A 0.000,B 0.000,C 90.000,E1 285.009} C_DIS
LIN {X -0.173,Y -426.840,Z 1515.579,A 0.000,B 0.000,C 90.000,E1 284.245} C_DIS
LIN {X 0.014,Y -429.886,Z 1515.574,A 0.000,B 0.000,C 90.000,E1 283.411} C_DIS
LIN {X -0.057,Y -431.497,Z 1515.572,A 0.000,B 0.000,C 90.000,E1 282.883} C_DIS
LIN {X -0.117,Y -432.698,Z 1515.569,A 0.000,B 0.000,C 90.000,E1 282.355} C_DIS
LIN {X -0.167,Y -433.445,Z 1515.566,A 0.000,B 0.000,C 90.000,E1 281.827} C_DIS
LIN {X 0.214,Y -433.686,Z 1515.563,A 0.000,B 0.000,C 90.000,E1 281.243} C_DIS
LIN {X 0.092,Y -433.436,Z 1515.560,A 0.000,B 0.000,C 90.000,E1 280.725} C_DIS
LIN {X 0.054,Y -432.611,Z 1515.557,A 0.000,B 0.000,C 90.000,E1 280.197} C_DIS
LIN {X 0.012,Y -431.193,Z 1515.554,A 0.000,B 0.000,C 90.000,E1 279.670} C_DIS
LIN {X -0.106,Y -429.108,Z 1515.551,A 0.000,B 0.000,C 90.000,E1 279.151} C_DIS
LIN {X -0.164,Y -426.314,Z 1515.548,A 0.000,B 0.000,C 90.000,E1 278.624} C_DIS
LIN {X 0.114,Y -422.647,Z 1515.545,A 0.000,B 0.000,C 90.000,E1 278.049} C_DIS
LIN {X -0.044,Y -418.015,Z 1515.542,A 0.000,B 0.000,C 90.000,E1 277.530} C_DIS
LIN {X -0.170,Y -412.336,Z 1515.539,A 0.000,B 0.000,C 90.000,E1 277.004} C_DIS
LIN {X 0.059,Y -406.302,Z 1515.536,A 0.000,B 0.000,C 90.000,E1 276.486} C_DIS
LIN {X -0.195,Y -400.049,Z 1515.534,A 0.000,B 0.000,C 90.000,E1 276.087} C_DIS
LIN {X -0.087,Y -393.657,Z 1515.531,A 0.000,B 0.000,C 90.000,E1 275.682} C_DIS
LIN {X -0.099,Y -387.143,Z 1515.530,A 0.000,B 0.000,C 90.000,E1 275.334} C_DIS
LIN {X -0.117,Y -377.283,Z 1515.527,A 0.000,B 0.000,C 90.000,E1 274.878} C_DIS
LIN {X 0.105,Y -361.408,Z 1515.523,A 0.000,B 0.000,C 90.000,E1 274.188} C_DIS
LIN {X -0.103,Y -348.661,Z 1515.521,A 0.000,B 0.000,C 90.000,E1 273.726} C_DIS
LIN {X -0.107,Y -338.757,Z 1515.519,A 0.000,B 0.000,C 90.000,E1 273.383} C_DIS
LIN {X 0.089,Y -328.806,Z 1515.517,A 0.000,B 0.000,C 90.000,E1 273.037} C_DIS
LIN {X -0.029,Y -315.276,Z 1515.515,A 0.000,B 0.000,C 90.000,E1 272.694} C_DIS
LIN {X -0.007,Y -304.128,Z 1515.514,A 0.000,B 0.000,C 90.000,E1 272.465} C_DIS
LIN {X -0.070,Y -296.151,Z 1515.513,A 0.000,B 0.000,C 90.000,E1 272.350} C_DIS
LIN {X -0.048,Y -286.556,Z 1515.512,A 0.000,B 0.000,C 90.000,E1 272.236} C_DIS
LIN {X -0.120,Y -276.122,Z 1515.512,A 0.000,B 0.000,C 90.000,E1 272.178} C_DIS
LIN {X 0.104,Y -272.314,Z 1515.512,A 0.000,B 0.000,C 90.000,E1 272.121} C_DIS
LIN {X 0.036,Y -181.241,Z 1515.512,A 0.000,B 0.000,C 90.000,E1 272.121} C_DIS
LIN {X 0.013,Y -181.576,Z 1515.502,A 0.000,B 0.000,C 90.000,E1 270.401} C_DIS
LIN {X -0.010,Y -180.906,Z 1515.474,A 0.000,B 0.000,C 90.000,E1 265.355} C_DIS
LIN {X 0.063,Y -180.680,Z 1515.469,A 0.000,B 0.000,C 90.000,E1 264.489} C_DIS
LIN {X -0.037,Y -178.762,Z 1515.441,A 0.000,B 0.000,C 90.000,E1 259.454} C_DIS
LIN {X 0.034,Y -175.809,Z 1515.413,A 0.000,B 0.000,C 90.000,E1 254.338} C_DIS
LIN {X 0.029,Y -171.996,Z 1515.385,A 0.000,B 0.000,C 90.000,E1 249.209} C_DIS
LIN {X 0.003,Y -171.408,Z 1515.380,A 0.000,B 0.000,C 90.000,E1 248.358} C_DIS
LIN {X 0.051,Y -167.649,Z 1515.356,A 0.000,B 0.000,C 90.000,E1 244.024} C_DIS
LIN {X 0.065,Y -166.312,Z 1515.346,A 0.000,B 0.000,C 90.000,E1 242.281} C_DIS
LIN {X 0.059,Y -163.055,Z 1515.327,A 0.000,B 0.000,C 90.000,E1 238.791} C_DIS
LIN {X 0.021,Y -160.990,Z 1515.312,A 0.000,B 0.000,C 90.000,E1 236.167} C_DIS
LIN {X -0.003,Y -157.737,Z 1515.292,A 0.000,B 0.000,C 90.000,E1 232.637} C_DIS
LIN {X -0.064,Y -155.776,Z 1515.278,A 0.000,B 0.000,C 90.000,E1 229.989} C_DIS
LIN {X -0.009,Y -152.031,Z 1515.253,A 0.000,B 0.000,C 90.000,E1 225.486} C_DIS
LIN {X 0.009,Y -150.279,Z 1515.238,A 0.000,B 0.000,C 90.000,E1 222.771} C_DIS
LIN {X 0.026,Y -147.029,Z 1515.212,A 0.000,B 0.000,C 90.000,E1 218.222} C_DIS
LIN {X -0.071,Y -145.610,Z 1515.197,A 0.000,B 0.000,C 90.000,E1 215.518} C_DIS
LIN {X 0.051,Y -142.996,Z 1515.172,A 0.000,B 0.000,C 90.000,E1 210.875} C_DIS
LIN {X -0.014,Y -141.622,Z 1515.151,A 0.000,B 0.000,C 90.000,E1 207.206} C_DIS
LIN {X 0.042,Y -139.432,Z 1515.115,A 0.000,B 0.000,C 90.000,E1 200.684} C_DIS
LIN {X -0.034,Y -139.163,Z 1515.105,A 0.000,B 0.000,C 90.000,E1 198.852} C_DIS
LIN {X 0.002,Y -138.341,Z 1515.058,A 0.000,B 0.000,C 90.000,E1 190.433} C_DIS
LIN {X 0.010,Y -139.478,Z 1515.006,A 0.000,B 0.000,C 90.000,E1 181.088} C_DIS
LIN {X -0.050,Y -141.064,Z 1514.975,A 0.000,B 0.000,C 90.000,E1 175.527} C_DIS
LIN {X 0.045,Y -142.437,Z 1514.960,A 0.000,B 0.000,C 90.000,E1 172.704} C_DIS
LIN {X -0.036,Y -144.676,Z 1514.934,A 0.000,B 0.000,C 90.000,E1 168.117} C_DIS
LIN {X -0.052,Y -147.264,Z 1514.913,A 0.000,B 0.000,C 90.000,E1 164.448} C_DIS
LIN {X -0.035,Y -150.581,Z 1514.888,A 0.000,B 0.000,C 90.000,E1 159.880} C_DIS
LIN {X 0.043,Y -154.052,Z 1514.868,A 0.000,B 0.000,C 90.000,E1 156.230} C_DIS
LIN {X -0.030,Y -157.470,Z 1514.848,A 0.000,B 0.000,C 90.000,E1 152.666} C_DIS
LIN {X 0.057,Y -161.693,Z 1514.828,A 0.000,B 0.000,C 90.000,E1 149.076} C_DIS
LIN {X -0.065,Y -165.887,Z 1514.809,A 0.000,B 0.000,C 90.000,E1 145.595} C_DIS
LIN {X -0.075,Y -170.869,Z 1514.789,A 0.000,B 0.000,C 90.000,E1 142.110} C_DIS
LIN {X -0.028,Y -175.737,Z 1514.770,A 0.000,B 0.000,C 90.000,E1 138.647} C_DIS
LIN {X -0.038,Y -181.347,Z 1514.751,A 0.000,B 0.000,C 90.000,E1 135.243} C_DIS
LIN {X 0.096,Y -186.837,Z 1514.733,A 0.000,B 0.000,C 90.000,E1 131.838} C_DIS
LIN {X 0.049,Y -191.424,Z 1514.719,A 0.000,B 0.000,C 90.000,E1 129.358} C_DIS
LIN {X -0.018,Y -197.274,Z 1514.700,A 0.000,B 0.000,C 90.000,E1 126.091} C_DIS
LIN {X 0.018,Y -200.552,Z 1514.691,A 0.000,B 0.000,C 90.000,E1 124.452} C_DIS
LIN {X 0.036,Y -202.205,Z 1514.686,A 0.000,B 0.000,C 90.000,E1 123.499} C_DIS
LIN {X 0.020,Y -316.177,Z 1514.686,A 0.000,B 0.000,C 90.000,E1 123.499} C_DIS
LIN {X 0.053,Y -318.626,Z 1514.686,A 0.000,B 0.000,C 90.000,E1 123.452} C_DIS
LIN {X -0.080,Y -324.237,Z 1514.684,A 0.000,B 0.000,C 90.000,E1 123.166} C_DIS
LIN {X 0.058,Y -327.224,Z 1514.682,A 0.000,B 0.000,C 90.000,E1 122.832} C_DIS
LIN {X 0.058,Y -329.227,Z 1514.681,A 0.000,B 0.000,C 90.000,E1 122.546} C_DIS
LIN {X 0.057,Y -330.795,Z 1514.679,A 0.000,B 0.000,C 90.000,E1 122.260} C_DIS
LIN {X -0.172,Y -333.328,Z 1514.676,A 0.000,B 0.000,C 90.000,E1 121.671} C_DIS
LIN {X 0.161,Y -344.541,Z 1514.660,A 0.000,B 0.000,C 90.000,E1 118.821} C_DIS
LIN {X 0.018,Y -357.155,Z 1514.645,A 0.000,B 0.000,C 90.000,E1 116.104} C_DIS
LIN {X -0.095,Y -371.270,Z 1514.630,A 0.000,B 0.000,C 90.000,E1 113.439} C_DIS
LIN {X -0.048,Y -385.182,Z 1514.617,A 0.000,B 0.000,C 90.000,E1 111.099} C_DIS
LIN {X 0.224,Y -400.475,Z 1514.604,A 0.000,B 0.000,C 90.000,E1 108.779} C_DIS
LIN {X 0.124,Y -417.256,Z 1514.592,A 0.000,B 0.000,C 90.000,E1 106.567} C_DIS
LIN {X 0.024,Y -435.643,Z 1514.580,A 0.000,B 0.000,C 90.000,E1 104.411} C_DIS
LIN {X -0.132,Y -455.411,Z 1514.569,A 0.000,B 0.000,C 90.000,E1 102.355} C_DIS
LIN {X -0.045,Y -475.782,Z 1514.558,A 0.000,B 0.000,C 90.000,E1 100.433} C_DIS
LIN {X 0.011,Y -491.281,Z 1514.551,A 0.000,B 0.000,C 90.000,E1 99.095} C_DIS
LIN {X 0.186,Y -493.209,Z 1514.549,A 0.000,B 0.000,C 90.000,E1 98.859} C_DIS
LIN {X 0.094,Y -494.877,Z 1514.548,A 0.000,B 0.000,C 90.000,E1 98.624} C_DIS
LIN {X -0.073,Y -496.122,Z 1514.547,A 0.000,B 0.000,C 90.000,E1 98.398} C_DIS
LIN {X 0.249,Y -497.635,Z 1514.544,A 0.000,B 0.000,C 90.000,E1 97.871} C_DIS
LIN {X 0.014,Y -498.080,Z 1514.541,A 0.000,B 0.000,C 90.000,E1 97.409} C_DIS
LIN {X -0.211,Y -497.528,Z 1514.538,A 0.000,B 0.000,C 90.000,E1 96.947} C_DIS
LIN {X 0.060,Y -495.895,Z 1514.536,A 0.000,B 0.000,C 90.000,E1 96.429} C_DIS
LIN {X -0.079,Y -494.580,Z 1514.534,A 0.000,B 0.000,C 90.000,E1 96.201} C_DIS
LIN {X 0.147,Y -484.746,Z 1514.526,A 0.000,B 0.000,C 90.000,E1 94.702} C_DIS
LIN {X 0.131,Y -475.668,Z 1514.518,A 0.000,B 0.000,C 90.000,E1 93.212} C_DIS
LIN {X 0.172,Y -467.612,Z 1514.511,A 0.000,B 0.000,C 90.000,E1 91.949} C_DIS
LIN {X 0.087,Y -459.139,Z 1514.504,A 0.000,B 0.000,C 90.000,E1 90.688} C_DIS
LIN {X 0.092,Y -448.581,Z 1514.495,A 0.000,B 0.000,C 90.000,E1 89.141} C_DIS
LIN {X 0.192,Y -439.661,Z 1514.488,A 0.000,B 0.000,C 90.000,E1 87.822} C_DIS
LIN {X 0.009,Y -426.729,Z 1514.478,A 0.000,B 0.000,C 90.000,E1 85.988} C_DIS
LIN {X 0.049,Y -413.889,Z 1514.467,A 0.000,B 0.000,C 90.000,E1 84.090} C_DIS
LIN {X -0.129,Y -401.086,Z 1514.457,A 0.000,B 0.000,C 90.000,E1 82.186} C_DIS
LIN {X 0.067,Y -381.475,Z 1514.439,A 0.000,B 0.000,C 90.000,E1 79.050} C_DIS
LIN {X -0.130,Y -364.767,Z 1514.423,A 0.000,B 0.000,C 90.000,E1 76.172} C_DIS
LIN {X -0.199,Y -353.444,Z 1514.411,A 0.000,B 0.000,C 90.000,E1 74.102} C_DIS
LIN {X 0.030,Y -340.646,Z 1514.398,A 0.000,B 0.000,C 90.000,E1 71.638} C_DIS
LIN {X 0.044,Y -328.122,Z 1514.384,A 0.000,B 0.000,C 90.000,E1 69.156} C_DIS
LIN {X 0.035,Y -314.749,Z 1514.368,A 0.000,B 0.000,C 90.000,E1 66.305} C_DIS
LIN {X -0.066,Y -300.531,Z 1514.350,A 0.000,B 0.000,C 90.000,E1 63.076} C_DIS
LIN {X -0.026,Y -289.630,Z 1514.336,A 0.000,B 0.000,C 90.000,E1 60.411} C_DIS
LIN {X -0.066,Y -279.118,Z 1514.321,A 0.000,B 0.000,C 90.000,E1 57.709} C_DIS
LIN {X 0.170,Y -268.867,Z 1514.305,A 0.000,B 0.000,C 90.000,E1 54.895} C_DIS
LIN {X -0.038,Y -260.117,Z 1514.292,A 0.000,B 0.000,C 90.000,E1 52.477} C_DIS
LIN {X 0.098,Y -249.378,Z 1514.274,A 0.000,B 0.000,C 90.000,E1 49.218} C_DIS
LIN {X 0.076,Y -240.497,Z 1514.257,A 0.000,B 0.000,C 90.000,E1 46.296} C_DIS
LIN {X 0.019,Y -232.317,Z 1514.241,A 0.000,B 0.000,C 90.000,E1 43.338} C_DIS
LIN {X -0.049,Y -224.909,Z 1514.224,A 0.000,B 0.000,C 90.000,E1 40.334} C_DIS
LIN {X 0.067,Y -218.303,Z 1514.207,A 0.000,B 0.000,C 90.000,E1 37.237} C_DIS
LIN {X 0.093,Y -212.376,Z 1514.190,A 0.000,B 0.000,C 90.000,E1 34.119} C_DIS
LIN {X -0.016,Y -205.843,Z 1514.168,A 0.000,B 0.000,C 90.000,E1 30.207} C_DIS
LIN {X -0.091,Y -200.053,Z 1514.146,A 0.000,B 0.000,C 90.000,E1 26.232} C_DIS
LIN {X 0.025,Y -195.163,Z 1514.123,A 0.000,B 0.000,C 90.000,E1 22.153} C_DIS
LIN {X 0.055,Y -191.046,Z 1514.100,A 0.000,B 0.000,C 90.000,E1 18.055} C_DIS
LIN {X -0.007,Y -187.044,Z 1514.073,A 0.000,B 0.000,C 90.000,E1 13.119} C_DIS
LIN {X -0.035,Y -183.722,Z 1514.041,A 0.000,B 0.000,C 90.000,E1 7.296} C_DIS
LIN {X 0.086,Y -181.744,Z 1513.988,A 0.000,B 0.000,C 90.000,E1 357.822} C_DIS
LIN {X -0.043,Y -183.196,Z 1513.941,A 0.000,B 0.000,C 90.000,E1 349.454} C_DIS
LIN {X 0.073,Y -186.200,Z 1513.909,A 0.000,B 0.000,C 90.000,E1 343.559} C_DIS
LIN {X 0.006,Y -190.018,Z 1513.881,A 0.000,B 0.000,C 90.000,E1 338.592} C_DIS
LIN {X 0.044,Y -194.226,Z 1513.858,A 0.000,B 0.000,C 90.000,E1 334.460} C_DIS
LIN {X 0.034,Y -199.304,Z 1513.836,A 0.000,B 0.000,C 90.000,E1 330.383} C_DIS
LIN {X -0.021,Y -204.125,Z 1513.818,A 0.000,B 0.000,C 90.000,E1 327.168} C_DIS
LIN {X -0.086,Y -209.633,Z 1513.800,A 0.000,B 0.000,C 90.000,E1 323.989} C_DIS
LIN {X 0.018,Y -215.922,Z 1513.782,A 0.000,B 0.000,C 90.000,E1 320.803} C_DIS
LIN {X -0.083,Y -223.015,Z 1513.765,A 0.000,B 0.000,C 90.000,E1 317.715} C_DIS
LIN {X 0.131,Y -231.039,Z 1513.748,A 0.000,B 0.000,C 90.000,E1 314.595} C_DIS
LIN {X -0.037,Y -238.893,Z 1513.733,A 0.000,B 0.000,C 90.000,E1 312.000} C_DIS
LIN {X -0.022,Y -247.750,Z 1513.719,A 0.000,B 0.000,C 90.000,E1 309.402} C_DIS
LIN {X 0.022,Y -254.823,Z 1513.709,A 0.000,B 0.000,C 90.000,E1 307.569} C_DIS
LIN {X -0.018,Y -261.192,Z 1513.701,A 0.000,B 0.000,C 90.000,E1 306.137} C_DIS
LIN {X 0.085,Y -268.226,Z 1513.693,A 0.000,B 0.000,C 90.000,E1 304.692} C_DIS
LIN {X 0.062,Y -276.011,Z 1513.685,A 0.000,B 0.000,C 90.000,E1 303.293} C_DIS
LIN {X -0.098,Y -288.984,Z 1513.674,A 0.000,B 0.000,C 90.000,E1 301.258} C_DIS
LIN {X 0.092,Y -303.323,Z 1513.662,A 0.000,B 0.000,C 90.000,E1 299.205} C_DIS
LIN {X 0.050,Y -324.471,Z 1513.648,A 0.000,B 0.000,C 90.000,E1 296.616} C_DIS
LIN {X 0.067,Y -345.840,Z 1513.635,A 0.000,B 0.000,C 90.000,E1 294.259} C_DIS
LIN {X 0.027,Y -361.890,Z 1513.625,A 0.000,B 0.000,C 90.000,E1 292.589} C_DIS
LIN {X 0.156,Y -372.568,Z 1513.619,A 0.000,B 0.000,C 90.000,E1 291.461} C_DIS
LIN {X -0.047,Y -380.448,Z 1513.615,A 0.000,B 0.000,C 90.000,E1 290.663} C_DIS
LIN {X 0.074,Y -390.706,Z 1513.609,A 0.000,B 0.000,C 90.000,E1 289.523} C_DIS
LIN {X 0.096,Y -398.012,Z 1513.604,A 0.000,B 0.000,C 90.000,E1 288.671} C_DIS
LIN {X 0.142,Y -404.971,Z 1513.599,A 0.000,B 0.000,C 90.000,E1 287.819} C_DIS
LIN {X 0.134,Y -411.270,Z 1513.594,A 0.000,B 0.000,C 90.000,E1 286.985} C_DIS
LIN {X -0.218,Y -416.893,Z 1513.590,A 0.000,B 0.000,C 90.000,E1 286.205} C_DIS
LIN {X -0.118,Y -421.785,Z 1513.585,A 0.000,B 0.000,C 90.000,E1 285.371} C_DIS
LIN {X 0.024,Y -425.852,Z 1513.581,A 0.000,B 0.000,C 90.000,E1 284.537} C_DIS
LIN {X -0.066,Y -428.172,Z 1513.578,A 0.000,B 0.000,C 90.000,E1 284.008} C_DIS
LIN {X -0.041,Y -430.199,Z 1513.575,A 0.000,B 0.000,C 90.000,E1 283.467} C_DIS
LIN {X -0.112,Y -431.803,Z 1513.572,A 0.000,B 0.000,C 90.000,E1 282.939} C_DIS
LIN {X -0.172,Y -433.050,Z 1513.569,A 0.000,B 0.000,C 90.000,E1 282.411} C_DIS
LIN {X 0.203,Y -433.888,Z 1513.566,A 0.000,B 0.000,C 90.000,E1 281.827} C_DIS
LIN {X 0.161,Y -434.213,Z 1513.563,A 0.000,B 0.000,C 90.000,E1 281.299} C_DIS
LIN {X 0.041,Y -434.013,Z 1513.560,A 0.000,B 0.000,C 90.000,E1 280.782} C_DIS
LIN {X 0.006,Y -433.257,Z 1513.557,A 0.000,B 0.000,C 90.000,E1 280.254} C_DIS
LIN {X -0.033,Y -431.955,Z 1513.554,A 0.000,B 0.000,C 90.000,E1 279.726} C_DIS
LIN {X -0.149,Y -429.952,Z 1513.551,A 0.000,B 0.000,C 90.000,E1 279.208} C_DIS
LIN {X 0.036,Y -428.705,Z 1513.550,A 0.000,B 0.000,C 90.000,E1 278.916} C_DIS
LIN {X -0.092,Y -425.554,Z 1513.547,A 0.000,B 0.000,C 90.000,E1 278.398} C_DIS
LIN {X -0.176,Y -421.541,Z 1513.544,A 0.000,B 0.000,C 90.000,E1 277.871} C_DIS
LIN {X 0.075,Y -416.552,Z 1513.541,A 0.000,B 0.000,C 90.000,E1 277.296} C_DIS
LIN {X 0.079,Y -410.732,Z 1513.538,A 0.000,B 0.000,C 90.000,E1 276.777} C_DIS
LIN {X 0.049,Y -404.639,Z 1513.535,A 0.000,B 0.000,C 90.000,E1 276.315} C_DIS
LIN {X -0.041,Y -398.254,Z 1513.533,A 0.000,B 0.000,C 90.000,E1 275.910} C_DIS
LIN {X 0.113,Y -391.774,Z 1513.531,A 0.000,B 0.000,C 90.000,E1 275.511} C_DIS
LIN {X 0.177,Y -385.197,Z 1513.529,A 0.000,B 0.000,C 90.000,E1 275.163} C_DIS
LIN {X -0.101,Y -375.236,Z 1513.526,A 0.000,B 0.000,C 90.000,E1 274.759} C_DIS
LIN {X -0.175,Y -359.508,Z 1513.523,A 0.000,B 0.000,C 90.000,E1 274.131} C_DIS
LIN {X 0.057,Y -346.836,Z 1513.520,A 0.000,B 0.000,C 90.000,E1 273.612} C_DIS
LIN {X 0.148,Y -333.559,Z 1513.518,A 0.000,B 0.000,C 90.000,E1 273.154} C_DIS
LIN {X -0.070,Y -320.097,Z 1513.516,A 0.000,B 0.000,C 90.000,E1 272.808} C_DIS
LIN {X -0.058,Y -313.121,Z 1513.515,A 0.000,B 0.000,C 90.000,E1 272.636} C_DIS
LIN {X -0.006,Y -301.057,Z 1513.513,A 0.000,B 0.000,C 90.000,E1 272.407} C_DIS
LIN {X -0.034,Y -292.588,Z 1513.513,A 0.000,B 0.000,C 90.000,E1 272.293} C_DIS
LIN {X -0.080,Y -278.706,Z 1513.512,A 0.000,B 0.000,C 90.000,E1 272.178} C_DIS
LIN {X 0.091,Y -271.102,Z 1513.512,A 0.000,B 0.000,C 90.000,E1 272.121} C_DIS
LIN {X 0.026,Y -181.241,Z 1513.512,A 0.000,B 0.000,C 90.000,E1 272.121} C_DIS
LIN {X 0.035,Y -181.575,Z 1513.502,A 0.000,B 0.000,C 90.000,E1 270.401} C_DIS
LIN {X 0.012,Y -180.906,Z 1513.474,A 0.000,B 0.000,C 90.000,E1 265.355} C_DIS
LIN {X 0.086,Y -180.684,Z 1513.469,A 0.000,B 0.000,C 90.000,E1 264.489} C_DIS
LIN {X -0.016,Y -178.767,Z 1513.441,A 0.000,B 0.000,C 90.000,E1 259.454} C_DIS
LIN {X 0.056,Y -175.814,Z 1513.413,A 0.000,B 0.000,C 90.000,E1 254.338} C_DIS
LIN {X 0.049,Y -172.000,Z 1513.385,A 0.000,B 0.000,C 90.000,E1 249.209} C_DIS
LIN {X 0.024,Y -171.415,Z 1513.380,A 0.000,B 0.000,C 90.000,E1 248.358} C_DIS
LIN {X 0.072,Y -167.654,Z 1513.356,A 0.000,B 0.000,C 90.000,E1 244.024} C_DIS
LIN {X 0.086,Y -166.319,Z 1513.346,A 0.000,B 0.000,C 90.000,E1 242.281} C_DIS
LIN {X -0.005,Y -163.060,Z 1513.327,A 0.000,B 0.000,C 90.000,E1 238.820} C_DIS
LIN {X 0.041,Y -160.997,Z 1513.312,A 0.000,B 0.000,C 90.000,E1 236.167} C_DIS
LIN {X 0.017,Y -157.744,Z 1513.292,A 0.000,B 0.000,C 90.000,E1 232.637} C_DIS
LIN {X -0.045,Y -155.782,Z 1513.278,A 0.000,B 0.000,C 90.000,E1 229.989} C_DIS
LIN {X 0.011,Y -152.036,Z 1513.253,A 0.000,B 0.000,C 90.000,E1 225.486} C_DIS
LIN {X 0.028,Y -150.284,Z 1513.238,A 0.000,B 0.000,C 90.000,E1 222.771} C_DIS
LIN {X -0.046,Y -147.034,Z 1513.212,A 0.000,B 0.000,C 90.000,E1 218.257} C_DIS
LIN {X -0.052,Y -145.614,Z 1513.197,A 0.000,B 0.000,C 90.000,E1 215.518} C_DIS
LIN {X -0.053,Y -142.999,Z 1513.172,A 0.000,B 0.000,C 90.000,E1 210.924} C_DIS
LIN {X 0.004,Y -141.626,Z 1513.151,A 0.000,B 0.000,C 90.000,E1 207.206} C_DIS
LIN {X -0.070,Y -139.433,Z 1513.115,A 0.000,B 0.000,C 90.000,E1 200.737} C_DIS
LIN {X -0.016,Y -139.165,Z 1513.105,A 0.000,B 0.000,C 90.000,E1 198.852} C_DIS
LIN {X 0.021,Y -138.340,Z 1513.058,A 0.000,B 0.000,C 90.000,E1 190.433} C_DIS
LIN {X 0.028,Y -139.477,Z 1513.006,A 0.000,B 0.000,C 90.000,E1 181.088} C_DIS
LIN {X -0.031,Y -141.060,Z 1512.975,A 0.000,B 0.000,C 90.000,E1 175.527} C_DIS
LIN {X 0.065,Y -142.433,Z 1512.960,A 0.000,B 0.000,C 90.000,E1 172.704} C_DIS
LIN {X -0.016,Y -144.671,Z 1512.934,A 0.000,B 0.000,C 90.000,E1 168.117} C_DIS
LIN {X -0.033,Y -147.258,Z 1512.914,A 0.000,B 0.000,C 90.000,E1 164.448} C_DIS
LIN {X -0.015,Y -150.575,Z 1512.888,A 0.000,B 0.000,C 90.000,E1 159.880} C_DIS
LIN {X 0.063,Y -154.046,Z 1512.868,A 0.000,B 0.000,C 90.000,E1 156.230} C_DIS
LIN {X -0.009,Y -157.463,Z 1512.848,A 0.000,B 0.000,C 90.000,E1 152.666} C_DIS
LIN {X -0.062,Y -161.683,Z 1512.828,A 0.000,B 0.000,C 90.000,E1 149.125} C_DIS
LIN {X -0.045,Y -165.878,Z 1512.809,A 0.000,B 0.000,C 90.000,E1 145.595} C_DIS
LIN {X -0.054,Y -170.857,Z 1512.789,A 0.000,B 0.000,C 90.000,E1 142.110} C_DIS
LIN {X -0.007,Y -175.726,Z 1512.770,A 0.000,B 0.000,C 90.000,E1 138.647} C_DIS
LIN {X -0.017,Y -181.338,Z 1512.751,A 0.000,B 0.000,C 90.000,E1 135.243} C_DIS
LIN {X 0.118,Y -186.825,Z 1512.733,A 0.000,B 0.000,C 90.000,E1 131.838} C_DIS
LIN {X 0.072,Y -191.413,Z 1512.719,A 0.000,B 0.000,C 90.000,E1 129.358} C_DIS
LIN {X 0.005,Y -197.261,Z 1512.701,A 0.000,B 0.000,C 90.000,E1 126.091} C_DIS
LIN {X -0.072,Y -200.539,Z 1512.692,A 0.000,B 0.000,C 90.000,E1 124.485} C_DIS
LIN {X -0.111,Y -202.139,Z 1512.686,A 0.000,B 0.000,C 90.000,E1 123.579} C_DIS
LIN {X 0.214,Y -315.542,Z 1512.686,A 0.000,B 0.000,C 90.000,E1 123.499} C_DIS
LIN {X 0.164,Y -316.783,Z 1512.686,A 0.000,B 0.000,C 90.000,E1 123.499} C_DIS
LIN {X -0.075,Y -321.635,Z 1512.685,A 0.000,B 0.000,C 90.000,E1 123.372} C_DIS
LIN {X 0.131,Y -324.041,Z 1512.684,A 0.000,B 0.000,C 90.000,E1 123.166} C_DIS
LIN {X 0.095,Y -327.287,Z 1512.682,A 0.000,B 0.000,C 90.000,E1 122.832} C_DIS
LIN {X 0.083,Y -329.258,Z 1512.681,A 0.000,B 0.000,C 90.000,E1 122.546} C_DIS
LIN {X 0.067,Y -330.801,Z 1512.679,A 0.000,B 0.000,C 90.000,E1 122.260} C_DIS
LIN {X -0.037,Y -334.478,Z 1512.674,A 0.000,B 0.000,C 90.000,E1 121.337} C_DIS
LIN {X -0.138,Y -345.844,Z 1512.659,A 0.000,B 0.000,C 90.000,E1 118.565} C_DIS
LIN {X 0.072,Y -358.615,Z 1512.643,A 0.000,B 0.000,C 90.000,E1 115.796} C_DIS
LIN {X 0.002,Y -372.908,Z 1512.629,A 0.000,B 0.000,C 90.000,E1 113.131} C_DIS
LIN {X 0.096,Y -386.985,Z 1512.616,A 0.000,B 0.000,C 90.000,E1 110.791} C_DIS
LIN {X -0.092,Y -402.458,Z 1512.603,A 0.000,B 0.000,C 90.000,E1 108.544} C_DIS
LIN {X -0.033,Y -419.433,Z 1512.591,A 0.000,B 0.000,C 90.000,E1 106.315} C_DIS
LIN {X 0.215,Y -438.029,Z 1512.579,A 0.000,B 0.000,C 90.000,E1 104.120} C_DIS
LIN {X 0.217,Y -457.904,Z 1512.567,A 0.000,B 0.000,C 90.000,E1 102.063} C_DIS
LIN {X 0.017,Y -478.342,Z 1512.557,A 0.000,B 0.000,C 90.000,E1 100.197} C_DIS
LIN {X 0.016,Y -491.234,Z 1512.551,A 0.000,B 0.000,C 90.000,E1 99.095} C_DIS
LIN {X 0.190,Y -493.148,Z 1512.549,A 0.000,B 0.000,C 90.000,E1 98.859} C_DIS
LIN {X 0.098,Y -494.805,Z 1512.548,A 0.000,B 0.000,C 90.000,E1 98.624} C_DIS
LIN {X -0.068,Y -496.042,Z 1512.547,A 0.000,B 0.000,C 90.000,E1 98.398} C_DIS
LIN {X 0.253,Y -497.543,Z 1512.544,A 0.000,B 0.000,C 90.000,E1 97.871} C_DIS
LIN {X 0.019,Y -497.975,Z 1512.541,A 0.000,B 0.000,C 90.000,E1 97.409} C_DIS
LIN {X -0.208,Y -497.413,Z 1512.538,A 0.000,B 0.000,C 90.000,E1 96.947} C_DIS
LIN {X 0.063,Y -495.767,Z 1512.536,A 0.000,B 0.000,C 90.000,E1 96.429} C_DIS
LIN {X -0.077,Y -494.446,Z 1512.534,A 0.000,B 0.000,C 90.000,E1 96.201} C_DIS
LIN {X -0.219,Y -486.156,Z 1512.528,A 0.000,B 0.000,C 90.000,E1 94.992} C_DIS
LIN {X 0.128,Y -475.528,Z 1512.518,A 0.000,B 0.000,C 90.000,E1 93.212} C_DIS
LIN {X 0.167,Y -467.479,Z 1512.511,A 0.000,B 0.000,C 90.000,E1 91.949} C_DIS
LIN {X 0.081,Y -459.027,Z 1512.504,A 0.000,B 0.000,C 90.000,E1 90.688} C_DIS
LIN {X 0.085,Y -448.483,Z 1512.495,A 0.000,B 0.000,C 90.000,E1 89.141} C_DIS
LIN {X -0.083,Y -437.745,Z 1512.487,A 0.000,B 0.000,C 90.000,E1 87.593} C_DIS
LIN {X 0.162,Y -424.843,Z 1512.476,A 0.000,B 0.000,C 90.000,E1 85.698} C_DIS
LIN {X 0.163,Y -412.056,Z 1512.466,A 0.000,B 0.000,C 90.000,E1 83.799} C_DIS
LIN {X -0.046,Y -399.270,Z 1512.455,A 0.000,B 0.000,C 90.000,E1 81.894} C_DIS
LIN {X 0.087,Y -379.784,Z 1512.438,A 0.000,B 0.000,C 90.000,E1 78.757} C_DIS
LIN {X -0.160,Y -363.185,Z 1512.421,A 0.000,B 0.000,C 90.000,E1 75.880} C_DIS
LIN {X 0.176,Y -351.882,Z 1512.410,A 0.000,B 0.000,C 90.000,E1 73.740} C_DIS
LIN {X 0.034,Y -339.094,Z 1512.396,A 0.000,B 0.000,C 90.000,E1 71.329} C_DIS
LIN {X 0.012,Y -326.608,Z 1512.382,A 0.000,B 0.000,C 90.000,E1 68.847} C_DIS
LIN {X 0.032,Y -314.754,Z 1512.368,A 0.000,B 0.000,C 90.000,E1 66.305} C_DIS
LIN {X -0.070,Y -300.525,Z 1512.350,A 0.000,B 0.000,C 90.000,E1 63.076} C_DIS
LIN {X -0.030,Y -289.649,Z 1512.336,A 0.000,B 0.000,C 90.000,E1 60.411} C_DIS
LIN {X -0.069,Y -279.172,Z 1512.321,A 0.000,B 0.000,C 90.000,E1 57.709} C_DIS
LIN {X 0.169,Y -268.981,Z 1512.305,A 0.000,B 0.000,C 90.000,E1 54.895} C_DIS
LIN {X -0.037,Y -260.266,Z 1512.292,A 0.000,B 0.000,C 90.000,E1 52.477} C_DIS
LIN {X 0.103,Y -249.579,Z 1512.274,A 0.000,B 0.000,C 90.000,E1 49.218} C_DIS
LIN {X 0.087,Y -240.720,Z 1512.257,A 0.000,B 0.000,C 90.000,E1 46.296} C_DIS
LIN {X 0.036,Y -232.570,Z 1512.241,A 0.000,B 0.000,C 90.000,E1 43.338} C_DIS
